	E_SequenceState.State_Active:
		//ProcessingQueue einmal durchlaufen
		fbProcessingQueue.M_SetCurrentToHead();
		REPEAT
			pStep := fbProcessingQueue.M_Get();
			IF pStep > 0 THEN
				CASE pStep^.eState OF
					E_StepState.STEPSTATUS_InQueue:
						nInfo := 0;
						//sind alle Bedingungen für eine Ausführung erfüllt?
						pStep^.bActionResultIsValid := FALSE;
						IF pStep^.pCondi > 0 THEN
							nCondiCheckResult := pStep^.pCondi^.M_Check(1);
							IF nCondiCheckResult.0 THEN
								//Hier checken, ob die Action einen Move mit Pipette beinhaltet
								//Wenn ja, dann checken, ob ZSensor mounted -> entsprechend Interaktion senden
								IF nCondiCheckResult.1 THEN //Cancel (Vergleich CondiStepResult negativ)
									//Step aus ProcessingQueue entfernen
									pStep^.bFollowerInQueue := FALSE;
									fbProcessingQueue.M_Remove(pStep);
									M_ChangeStepState(pStep, E_StepState.STEPSTATUS_Idle);
									fbSequenceInfo.M_AddTail(nId,eCurrentState,pStep);
								ELSE
									IF pStep^.stActionData.eAction = E_Action.ACTION_CounterStep THEN
										IF NOT pStep^.bFollowerInQueue THEN	//Follower in ProcessingQueue eintragen
											pStep^.bFollowerInQueue := TRUE;
											REPEAT
												pFollowStep := M_ReadFollowerStep(pStep);
												IF pFollowStep > 0 THEN
													fbProcessingQueue.M_Add(pFollowStep);
													M_ChangeStepState(pFollowStep,E_StepState.STEPSTATUS_InQueue);
													M_ChangeStepInfo(pFollowStep,0);
													fbSequenceInfo.M_AddTail(nId,eCurrentState,pFollowStep);
												END_IF
											UNTIL (pFollowStep = 0)
											END_REPEAT
										END_IF
										
										IF pStep^.stActionData.aParams[1] = 0 THEN //Set
											pStep^.nActionResult := pStep^.stActionData.aParams[2];
										ELSIF pStep^.stActionData.aParams[1] = 1 THEN //Add
											pStep^.nActionResult := pStep^.nActionResult + pStep^.stActionData.aParams[2];
										END_IF
										
										//Provisorium
										nCounter := pStep^.nActionResult;
										//Provisorium
										
										nInfo := pStep^.nActionResult;
										pStep^.bActionResultIsValid := TRUE;
										//Step aus ProcessingQueue entfernen
										pStep^.bFollowerInQueue := FALSE;
										fbProcessingQueue.M_Remove(pStep);
										M_ChangeStepState(pStep, E_StepState.STEPSTATUS_Ready);
										M_ChangeStepInfo(pStep,pStep^.nActionResult);
										fbSequenceInfo.M_AddTail(nId,eCurrentState,pStep);
									ELSIF pStep^.stActionData.eAction = E_Action.ACTION_PauseStep THEN //PauseStep führt keine Action aus
										M_ChangeStepState(pStep, E_StepState.STEPSTATUS_Active);
										fbSequenceInfo.M_AddTail(nId,eCurrentState,pStep);
									ELSE //Action ausführen
										M_ChangeStepState(pStep, E_StepState.STEPSTATUS_Active);
										IF pStep^.stActionData.eAction = E_Action.ACTION_MoveToTarget AND pStep^.stActionData.aParams[1] = E_TargetRef.TARGETREF_SequParaToArrayItem THEN
											pStep^.stActionData.aParams[2] := nSequParam;
										ELSIF pStep^.stActionData.eAction = E_Action.ACTION_RunSequence THEN
											pStep^.stActionData.aParams[2] := nCounter;
										END_IF
										stError.ErrorId := ActionDispacher.M_ExeAction(pStep^.stActionData, FALSE, nActionId=>pStep^.nActionId);
										fbSequenceInfo.M_AddTail(nId,eCurrentState,pStep);
									END_IF
								END_IF
							END_IF
						ELSE	//Step hat keine Condi
							M_ChangeStepState(pStep, E_StepState.STEPSTATUS_Active);
							IF pStep^.stActionData.eAction = E_Action.ACTION_CounterStep THEN
								IF NOT pStep^.bFollowerInQueue THEN	//Follower in ProcessingQueue eintragen
									pStep^.bFollowerInQueue := TRUE;
									REPEAT
										pFollowStep := M_ReadFollowerStep(pStep);
										IF pFollowStep > 0 THEN
											fbProcessingQueue.M_Add(pFollowStep);
											M_ChangeStepState(pFollowStep, E_StepState.STEPSTATUS_InQueue);
											M_ChangeStepInfo(pFollowStep,0);
											fbSequenceInfo.M_AddTail(nId,eCurrentState,pFollowStep);
										END_IF
									UNTIL (pFollowStep = 0)
									END_REPEAT
								END_IF
								
								IF pStep^.stActionData.aParams[1] = 0 THEN //Set
									pStep^.nActionResult := pStep^.stActionData.aParams[2];
								ELSIF pStep^.stActionData.aParams[1] = 1 THEN //Add
									pStep^.nActionResult := pStep^.nActionResult + pStep^.stActionData.aParams[2];
								END_IF
								
								//Provisorium
								nCounter := pStep^.nActionResult;
								//Provisorium
								
								pStep^.bActionResultIsValid := TRUE;
								//Step aus ProcessingQueue entfernen
								pStep^.bFollowerInQueue := FALSE;
								fbProcessingQueue.M_Remove(pStep);
								M_ChangeStepState(pStep, E_StepState.STEPSTATUS_Ready);
								M_ChangeStepInfo(pStep,pStep^.nActionResult);
								fbSequenceInfo.M_AddTail(nId,eCurrentState,pStep);
							ELSIF pStep^.stActionData.eAction = E_Action.ACTION_PauseStep THEN //PauseStep führt keine Action aus
								M_ChangeStepState(pStep, E_StepState.STEPSTATUS_Active);
								fbSequenceInfo.M_AddTail(nId,eCurrentState,pStep);
							ELSE //Action ausführen
								M_ChangeStepState(pStep, E_StepState.STEPSTATUS_Active);
								
								IF pStep^.stActionData.eAction = E_Action.ACTION_MoveToTarget AND pStep^.stActionData.aParams[1] = E_TargetRef.TARGETREF_SequParaToArrayItem THEN
									pStep^.stActionData.aParams[2] := nSequParam;
								ELSIF pStep^.stActionData.eAction = E_Action.ACTION_RunSequence THEN
									pStep^.stActionData.aParams[2] := nCounter;
								END_IF
								
								stError.ErrorId := ActionDispacher.M_ExeAction(pStep^.stActionData, FALSE, nActionId=>pStep^.nActionId);
								fbSequenceInfo.M_AddTail(nId,eCurrentState,pStep);
							END_IF
						END_IF
						
						IF stError.ErrorId > 0 THEN
							M_ChangeStepState(pStep, E_StepState.STEPSTATUS_Error);
							fbSequenceInfo.M_AddTail(nId,eCurrentState,pStep);
							bError := TRUE;
						END_IF
						
						
					E_StepState.STEPSTATUS_Active:
						IF NOT pStep^.bFollowerInQueue THEN	//Follower in ProcessingQueue eintragen
							pStep^.bFollowerInQueue := TRUE;
							REPEAT
								pFollowStep := M_ReadFollowerStep(pStep);
								IF pFollowStep > 0 THEN
									fbProcessingQueue.M_Add(pFollowStep);
									M_ChangeStepState(pFollowStep, E_StepState.STEPSTATUS_InQueue);
									M_ChangeStepInfo(pFollowStep,pFollowStep^.nActionResult);
									fbSequenceInfo.M_AddTail(nId,eCurrentState,pFollowStep);
								END_IF
							UNTIL (pFollowStep = 0)
							END_REPEAT
						END_IF
						
						IF pStep^.stActionData.eAction = E_Action.ACTION_PauseStep THEN
							eCurrentState := E_SequenceState.State_PauseRequest;
							EXIT;
						ELSE
							//Action-Status abfragen
							IF nId = 1 THEN
								nId := 1;
							END_IF
							eActionStatus := ActionDispacher.M_GetActionStatus(pStep^.nActionId,nProgress=>nInfo);
							M_ChangeStepInfo(pStep, nInfo); 
							IF eActionStatus = E_ActionStatus.ACTIONSTATUS_Ready OR eActionStatus = E_ActionStatus.ACTIONSTATUS_Idle THEN //Action nicht mehr aktiv
								//Es gibt momentan genau eine Action, welche nach ihrer Abarbeitung die Sequence in Pause versetzt (DispenseTest)
								//Rückmeldung aus ActionDispacher
								//PauseRequest beim ActionDispacher gesetzt?
								//Delay bis Fertigmeldung
								M_ChangeStepState(pStep, E_StepState.STEPSTATUS_Ready);
								pStep^.bFollowerInQueue := FALSE;
								fbProcessingQueue.M_Remove(pStep);
								IF ActionDispacher.P_bLastActionResult THEN
									pStep^.bActionResultIsValid := TRUE;
									pStep^.nActionResult := ActionDispacher.P_nLastActionResult;
									M_ChangeStepInfo(pStep, pStep^.nActionResult);
									ActionDispacher.P_bLastActionResult := FALSE;
								END_IF
								IF ActionDispacher.P_bPauseRequestIntern THEN
									ActionDispacher.P_bPauseRequestIntern := FALSE;
									eCurrentState := E_SequenceState.State_PauseRequest;
									fbSequenceInfo.M_AddTail(nId,eCurrentState,pStep);
									EXIT;
								END_IF
							ELSIF eActionStatus = E_ActionStatus.ACTIONSTATUS_Pause THEN
								//Tritt auf, wenn Action intern auf Pause gesetzt werden (z.B. Untersequenzen, welche einen Pause-Step beinhalten)
								//->Seq. selber in Pause versetzen
								M_ChangeStepState(pStep, E_StepState.STEPSTATUS_Pause);
								eCurrentState := E_SequenceState.State_Pause;
								fbSequenceInfo.M_AddTail(nId,eCurrentState,pStep);
								EXIT;
							ELSIF eActionStatus = E_ActionStatus.ACTIONSTATUS_Error THEN //Action hat Error verursacht
								M_ChangeStepState(pStep, E_StepState.STEPSTATUS_Error);
								fbProcessingQueue.M_Remove(pStep);
								bError := TRUE;
							END_IF
							//Nur melden, wenn sich am jeweiligem Step etwas geändert hat
							//Diese Info kann nur im Step selber stehen.
							fbSequenceInfo.M_AddTail(nId,eCurrentState,pStep);
						END_IF
				END_CASE
			END_IF
		UNTIL (pStep = 0)
		END_REPEAT
		//Sequence ist abgearbeitet, wenn der letzte Step ready
		IF fbProcessingQueue.P_bEmpty THEN
			eCurrentState := E_SequenceState.State_Ready;
		END_IF
		
	E_SequenceState.State_PauseRequest:
		eCurrentState := E_SequenceState.State_Pause;
		//Active Steps in PauseRequest setzen
		//In diesem State wird solange verharrt, bis kein Step mehr in Active
		//ProcessingQueue einmal durchlaufen
		fbProcessingQueue.M_SetCurrentToHead();
		REPEAT
			pStep := fbProcessingQueue.M_Get();
			IF pStep > 0 THEN
				IF pStep^.eState = E_StepState.STEPSTATUS_Active THEN
					eCurrentState := E_SequenceState.State_PauseRequest; 
					CASE ActionDispacher.M_GetActionStatus(pStep^.nActionId,nProgress=>nInfo) OF
						E_ActionStatus.ACTIONSTATUS_Active:
							ActionDispacher.M_PauseAction(pStep^.nActionId);
						E_ActionStatus.ACTIONSTATUS_Pause:
							M_ChangeStepState(pStep, E_StepState.STEPSTATUS_Pause);
							fbSequenceInfo.M_AddTail(nId,eCurrentState,pStep);
						E_ActionStatus.ACTIONSTATUS_Ready:
							M_ChangeStepState(pStep, E_StepState.STEPSTATUS_Ready);
							pStep^.bFollowerInQueue := FALSE;
							fbProcessingQueue.M_Remove(pStep);
							fbSequenceInfo.M_AddTail(nId,eCurrentState,pStep);
							IF ActionDispacher.P_bLastActionResult THEN
								pStep^.bActionResultIsValid := TRUE;
								pStep^.nActionResult := ActionDispacher.P_nLastActionResult; 
								ActionDispacher.P_bLastActionResult := FALSE;
							END_IF
					END_CASE
				END_IF
			END_IF
		UNTIL (pStep = 0)
		END_REPEAT
	E_SequenceState.State_Pause:
		//Do nothing
	E_SequenceState.State_Continue:
		//Steps, die in Pause sind, fortsetzen
		fbProcessingQueue.M_SetCurrentToHead();
		REPEAT
			pStep := fbProcessingQueue.M_Get();
			IF pStep > 0 THEN
				IF pStep^.eState = E_StepState.STEPSTATUS_Pause THEN
					ActionDispacher.M_ContinueAction(pStep^.nActionId,nProgress=>nInfo);
					M_ChangeStepState(pStep, E_StepState.STEPSTATUS_Active);
					M_ChangeStepInfo(pStep, nInfo);
					fbSequenceInfo.M_AddTail(nId,eCurrentState,pStep);
				END_IF
			END_IF
		UNTIL (pStep = 0)
		END_REPEAT
		eCurrentState := E_SequenceState.State_Active;
	
	E_SequenceState.State_Ready:
		//Do nothing
	E_SequenceState.State_Cancel:
		//Alle aktiven Steps abbrechen
		//ProcessingQueue leeren
		//in Canceled gehen
		IF nCancelState = 0 THEN
			fbComplexAction.P_nDispenseTrials := 0;
			fbProcessingQueue.M_SetCurrentToHead();
			REPEAT
				pStep := fbProcessingQueue.M_Get();
				IF pStep > 0 THEN
					IF pStep^.eState = E_StepState.STEPSTATUS_Active OR pStep^.eState = E_StepState.STEPSTATUS_Pause THEN
						ActionDispacher.M_StopAction(pStep^.nActionId);
					END_IF
				END_IF
			UNTIL (pStep = 0)
			END_REPEAT
			nCancelState := 1;
		ELSIF nCancelState = 1 THEN
			eCurrentState := E_SequenceState.State_Canceled;	
			fbProcessingQueue.M_SetCurrentToHead();
			REPEAT
				pStep := fbProcessingQueue.M_Get();
				IF pStep > 0 THEN
					IF pStep^.eState = E_StepState.STEPSTATUS_Active OR pStep^.eState = E_StepState.STEPSTATUS_Pause THEN
						//kommt man hier an?
						//geht ActionStatus in Ready oder Idle?
						//eventuell mit Scope aufzeichnen
						IF ActionDispacher.M_GetActionStatus(pStep^.nActionId) <> E_ActionStatus.ACTIONSTATUS_Ready THEN
							eCurrentState := E_SequenceState.State_Cancel;
						END_IF
					END_IF
				END_IF
			UNTIL (pStep = 0)
			END_REPEAT			
		END_IF
END_CASE

IF eOldState <> eCurrentState THEN
	//Progress?
	fbSequenceInfo.M_AddTail(nId,eCurrentState,0);
	eOldState := eCurrentState;
END_IF

IF bError THEN
	fbComplexAction.P_nDispenseTrials := 0;
	stError.POU := POU_FB_Sequenece;
	fbErrorList.M_Add(stError);
	eCurrentState := E_SequenceState.State_Error;
	bError := FALSE;
END_IF

METHOD FB_init : BOOL
VAR_INPUT
	bInitRetains : BOOL; // if TRUE, the retain variables are initialized (warm start / cold start)
	bInCopyCode : BOOL;  // if TRUE, the instance afterwards gets moved into the copy code (online change)
	nNoOfSteps	: UINT;
END_VAR
fbStepList.FB_SetNoOfSteps(nNoOfSteps);
END_METHOD

METHOD M_AddCondi : ERRORID
VAR_INPUT
	refCmdData : REFERENCE TO  ST_CmdData;	
END_VAR
VAR
	eOperator : E_LogicOperator;
	pCondi : POINTER TO FB_CondiBase;
	pStep  : POINTER TO ST_Step; 
END_VAR
//checken, ob zugehörige /ProgramNr/StepNr vorhanden, dh. es muss schon eine Condition vorhanden sein, in die dann der
//Zeiger auf hinzuzufügende Condition eingetragen wird
pStep := fbStepList.M_Get(refCmdData.aHeader[0]);
IF pStep = 0 THEN
	M_AddCondi := E_ErrorIdCmd.ERRORID_StepNotExists;
	RETURN;
END_IF

IF pStep^.pCondi = 0 THEN	//Step besitzt noch keine Condition und kann deshalb keine zusätzliche bekommen
	M_AddCondi := E_ErrorIdCmd.ERRORID_StepHasNoBasicCondi;
	RETURN;
END_IF

eOperator := UINT_TO_USINT(refCmdData.aHeader[1]);

IF NOT (eOperator = E_LogicOperator.LOGIC_OP_AND OR eOperator = E_LogicOperator.LOGIC_OP_OR) THEN	//unzulässiger CondiOperator
	M_AddCondi := E_ErrorIdCmd.ERRORID_InvalidCondiOperator;
	RETURN;
END_IF

M_AddCondi := M_CreateCondi(pStep:= pStep, 
				eOperator:= eOperator, 
				eCondition:= DINT_TO_USINT(refCmdData.n32Data[0]), 
				nValue1:= refCmdData.n32Data[1], 
				nValue2:= refCmdData.n32Data[2], 
				nValue3:= refCmdData.n32Data[3], 
				pCondi=>pCondi);

IF M_AddCondi = 0 THEN
	pStep^.pCondi^.M_AddNext(pCondi);
END_IF
END_METHOD

METHOD M_AddStep : ERRORID
VAR_INPUT
	refCmdData : REFERENCE TO  ST_CmdData;
END_VAR

VAR
	stStep		: ST_Step;
	eCondition 	: E_Condition;
END_VAR
//Es werden nur Programmsätze mit zulässiger Action hinzugefügt
stStep.nStepNr := refCmdData.aHeader[0];
stStep.bStop := refCmdData.aHeader[1].0;
stStep.tDelay := UINT_TO_TIME(refCmdData.aHeader[2]);
stStep.stActionData.eAction := DINT_TO_UINT(refCmdData.n32Data[5]);
stStep.stActionData.nObject := DINT_TO_UINT(refCmdData.n32Data[6]);
stStep.bFollowerInQueue := FALSE;
stStep.bHasForerunner := FALSE;

//Basiscondtion hinzufügen
eCondition := DINT_TO_USINT(refCmdData.n32Data[0]);

M_AddStep := M_CreateCondi(pStep:= ADR(stStep), 
							eOperator:= E_LogicOperator.LOGIC_OP_AND,	//bei der ersten Condi immer "AND"
							eCondition:= eCondition, 
							nValue1:= refCmdData.n32Data[1], 
							nValue2:= refCmdData.n32Data[2], 
							nValue3:= refCmdData.n32Data[3], 
							pCondi=> stStep.pCondi);

IF M_AddStep > 0 THEN
	RETURN;
END_IF

CASE stStep.stActionData.eAction OF
	//BasicActions
	E_Action.ACTION_MoveXY, E_Action.ACTION_MoveZ, E_Action.ACTION_SetPressure, E_Action.ACTION_SetVacuum, E_Action.ACTION_SwitchPressure, 
	E_Action.ACTION_Heating, E_Action.ACTION_Cooling, E_Action.ACTION_Aspirate, E_Action.ACTION_Dispense, E_Action.ACTION_DispenseDrops, 
	E_Action.ACTION_InkSpin, E_Action.ACTION_Expose, E_Action.ACTION_InkOpClCover, E_Action.ACTION_ReactorOpCl, E_Action.ACTION_FillLiquid,
	E_Action.ACTION_EmptyLiquid, E_Action.ACTION_DilPrepare,E_Action.ACTION_Mix,E_Action.ACTION_MeasurepH,E_Action.ACTION_SetVoltage,
	E_Action.ACTION_SuckOff, E_Action.ACTION_BasicDispense, E_Action.ACTION_StirrCartridge,
	E_Action.ACTION_MoveLifter, E_Action.ACTION_TurnTo:
		//max 8 Parameter kopieren
		MEMCPY(ADR(stStep.stActionData.aParams),ADR(refCmdData.n32Data[7]),32);
	E_Action.ACTION_TakePicture:
		//1 Parameter kopieren
		MEMCPY(ADR(stStep.stActionData.aParams),ADR(refCmdData.n32Data[7]),4);
		//Parameter 2 wird mit SequenceID gefüllt und Parameter 3 wird mit StepNummer gefüllt
		stStep.stActionData.aParams[2] := UDINT_TO_DINT(nId);
		stStep.stActionData.aParams[3] := stStep.nStepNr;
	
	//ComplexActions
	E_Action.ACTION_MoveToTarget, E_Action.ACTION_ExchangePiece,E_Action.ACTION_OpenCloseFlipTube,E_Action.ACTION_InsertTool,
	E_Action.ACTION_DockTool:
		//Object muss ein MzTool sein
		IF fbObjectDirectory.M_ObjIsMzTool(stStep.stActionData.nObject) THEN
			stStep.stActionData.nTarget := DINT_TO_UINT(refCmdData.n32Data[7]);
			//Target checken
			IF fbObjectDirectory.M_ObjIsTarget(stStep.stActionData.nTarget) THEN
				//11 Parameter kopieren
				MEMCPY(ADR(stStep.stActionData.aParams),ADR(refCmdData.n32Data[8]),44);
			ELSE
				M_AddStep := E_ErrorIdCmd.ERRORID_UnsuitableTarget;
			END_IF
		ELSE
			M_AddStep := E_ErrorIdCmd.ERRORID_UnsuitableObject;
		END_IF

	E_Action.ACTION_TransferGas, E_Action.ACTION_TransferLiquid:
		//Object und Target müssen ein Luers sein
		IF fbObjectDirectory.M_GetObjType(stStep.stActionData.nObject) = E_ObjectType.OBJECTTYPE_Luer THEN
			stStep.stActionData.nTarget := DINT_TO_UINT(refCmdData.n32Data[7]);
			IF fbObjectDirectory.M_GetObjType(stStep.stActionData.nTarget) = E_ObjectType.OBJECTTYPE_Luer THEN
				//max. 3 Parameter kopieren
				MEMCPY(ADR(stStep.stActionData.aParams),ADR(refCmdData.n32Data[8]),12);
			ELSE
				M_AddStep := E_ErrorIdCmd.ERRORID_UnsuitableObject;
			END_IF
		ELSE
			M_AddStep := E_ErrorIdCmd.ERRORID_UnsuitableObject;
		END_IF
		
	E_Action.ACTION_TransferTray:
		IF fbObjectDirectory.M_ObjIsDevice(stStep.stActionData.nObject) THEN
			MEMCPY(ADR(stStep.stActionData.aParams),ADR(refCmdData.n32Data[8]),4);
		ELSE
			M_AddStep := E_ErrorIdCmd.ERRORID_UnsuitableObject;
		END_IF
	
	E_Action.ACTION_MeasureTool:
		//Object muss ein MzTool sein
		IF fbObjectDirectory.M_ObjIsMzTool(stStep.stActionData.nObject) THEN
			stStep.stActionData.nTarget := DINT_TO_UINT(refCmdData.n32Data[7]);
			MEMCPY(ADR(stStep.stActionData.aParams),ADR(refCmdData.n32Data[8]),12);
			//Target checken
			IF fbObjectDirectory.M_ObjIsTarget(stStep.stActionData.nTarget) THEN
				;
			ELSE
				M_AddStep := E_ErrorIdCmd.ERRORID_UnsuitableTarget;
			END_IF
		ELSE
			M_AddStep := E_ErrorIdCmd.ERRORID_UnsuitableObject;
		END_IF		
		
	E_Action.ACTION_CleanTip:
		//Object muss ein MzTool sein
		IF fbObjectDirectory.M_ObjIsMzTool(stStep.stActionData.nObject) THEN
			stStep.stActionData.nTarget := DINT_TO_UINT(refCmdData.n32Data[7]);
			//Target checken
			IF fbObjectDirectory.M_GetObjType(stStep.stActionData.nTarget) = E_ObjectType.OBJECTTYPE_TipCleaner THEN
				;
			ELSIF
				fbObjectDirectory.M_GetObjType(stStep.stActionData.nTarget) = E_ObjectType.OBJECTTYPE_TipCleanerGen2 THEN
				MEMCPY(ADR(stStep.stActionData.aParams[1]),ADR(refCmdData.n32Data[8]),16);
			ELSE
				M_AddStep := E_ErrorIdCmd.ERRORID_UnsuitableTarget;
			END_IF
		ELSE
			M_AddStep := E_ErrorIdCmd.ERRORID_UnsuitableObject;
		END_IF
		
	E_Action.ACTION_DryPip:
		//Object muss ein MzTool sein
		IF fbObjectDirectory.M_ObjIsMzTool(stStep.stActionData.nObject) THEN
			stStep.stActionData.nTarget := DINT_TO_UINT(refCmdData.n32Data[7]);
			//Target checken
			IF fbObjectDirectory.M_GetObjType(stStep.stActionData.nTarget) = E_ObjectType.OBJECTTYPE_DryPad THEN
				MEMCPY(ADR(stStep.stActionData.aParams[1]),ADR(refCmdData.n32Data[8]),8);
			ELSE
				M_AddStep := E_ErrorIdCmd.ERRORID_UnsuitableTarget;
			END_IF
		ELSE
			M_AddStep := E_ErrorIdCmd.ERRORID_UnsuitableObject;
		END_IF		
		
	E_Action.ACTION_WashTool:
		//Object muss eine Pipette sein
		IF fbObjectDirectory.M_GetObjType(stStep.stActionData.nObject) = E_ObjectType.OBJECTTYPE_PiezoPip OR
				fbObjectDirectory.M_GetObjType(stStep.stActionData.nObject) = E_ObjectType.OBJECTTYPE_PassivPip OR
				fbObjectDirectory.M_GetObjType(stStep.stActionData.nObject) = E_ObjectType.OBJECTTYPE_Luer OR
				fbObjectDirectory.M_GetObjType(stStep.stActionData.nObject) = E_ObjectType.OBJECTTYPE_SolenoidPip OR
				fbObjectDirectory.M_GetObjType(stStep.stActionData.nObject) = E_ObjectType.OBJECTTYPE_TitrationTool OR
				fbObjectDirectory.M_GetObjType(stStep.stActionData.nObject) = E_ObjectType.OBJECTTYPE_TwinPiezoHolder OR
				fbObjectDirectory.M_GetObjType(stStep.stActionData.nObject) = E_ObjectType.OBJECTTYPE_TriplePip THEN
			stStep.stActionData.nTarget := DINT_TO_UINT(refCmdData.n32Data[7]);
			//Target checken
			IF fbObjectDirectory.M_GetObjType(stStep.stActionData.nTarget) = E_ObjectType.OBJECTTYPE_WashStation THEN
				//5 Parameter kopieren
				MEMCPY(ADR(stStep.stActionData.aParams[1]),ADR(refCmdData.n32Data[8]),60);
			ELSE
				M_AddStep := E_ErrorIdCmd.ERRORID_UnsuitableTarget;
			END_IF
		ELSE
			M_AddStep := E_ErrorIdCmd.ERRORID_UnsuitableObject;
		END_IF
		
	E_Action.ACTION_DispenseTest:
		//Object muss eine PiezoPip
		IF (fbObjectDirectory.M_GetObjType(stStep.stActionData.nObject) = E_ObjectType.OBJECTTYPE_PiezoPip) OR
			(fbObjectDirectory.M_GetObjType(stStep.stActionData.nObject) = E_ObjectType.OBJECTTYPE_TwinPiezoHolder) THEN
			stStep.stActionData.nTarget := DINT_TO_UINT(refCmdData.n32Data[7]);
			//Target checken
			IF fbObjectDirectory.M_GetObjType(stStep.stActionData.nTarget) = E_ObjectType.OBJECTTYPE_Stroboscope THEN
				MEMCPY(ADR(stStep.stActionData.aParams[1]),ADR(refCmdData.n32Data[8]),8);
			ELSE
				M_AddStep := E_ErrorIdCmd.ERRORID_UnsuitableTarget;
			END_IF
		ELSE
			M_AddStep := E_ErrorIdCmd.ERRORID_UnsuitableObject;
		END_IF

	E_Action.ACTION_GetPipSample:
		//Object muss eine Pipette sein
		IF fbObjectDirectory.M_GetObjType(stStep.stActionData.nObject) = E_ObjectType.OBJECTTYPE_PiezoPip OR
				fbObjectDirectory.M_GetObjType(stStep.stActionData.nObject) = E_ObjectType.OBJECTTYPE_PassivPip OR
				fbObjectDirectory.M_GetObjType(stStep.stActionData.nObject) = E_ObjectType.OBJECTTYPE_SolenoidPip OR
				fbObjectDirectory.M_GetObjType(stStep.stActionData.nObject) = E_ObjectType.OBJECTTYPE_TwinPiezoHolder THEN
			stStep.stActionData.nTarget := DINT_TO_UINT(refCmdData.n32Data[7]);
			//Target checken
			IF fbObjectDirectory.M_GetObjType(stStep.stActionData.nTarget) = E_ObjectType.OBJECTTYPE_Mtp THEN
				//6 Parameter kopieren
				MEMCPY(ADR(stStep.stActionData.aParams[1]),ADR(refCmdData.n32Data[8]),24);		
			ELSE
				M_AddStep := E_ErrorIdCmd.ERRORID_UnsuitableTarget;
			END_IF
		ELSE
			M_AddStep := E_ErrorIdCmd.ERRORID_UnsuitableObject;
		END_IF
		
	E_Action.ACTION_StampDemolding:
		//Object muss ein StampSupport sein
		IF fbObjectDirectory.M_GetObjType(stStep.stActionData.nObject) = E_ObjectType.OBJECTTYPE_StampSupport THEN
			//6 Parameter kopieren
			MEMCPY(ADR(stStep.stActionData.aParams[1]),ADR(refCmdData.n32Data[7]),24);			
		ELSE
			M_AddStep := E_ErrorIdCmd.ERRORID_UnsuitableObject;
		END_IF
		
	E_Action.ACTION_StampInking:
		//Object muss ein StampSupport sein
		IF fbObjectDirectory.M_GetObjType(stStep.stActionData.nObject) = E_ObjectType.OBJECTTYPE_StampSupport THEN
			stStep.stActionData.nTarget := DINT_TO_UINT(refCmdData.n32Data[7]);
			//3 Parameter kopieren
			MEMCPY(ADR(stStep.stActionData.aParams[1]),ADR(refCmdData.n32Data[8]),12);
		ELSE	
			M_AddStep := E_ErrorIdCmd.ERRORID_UnsuitableObject;
		END_IF
		
	E_Action.ACTION_PickPutPowder:
		//Object kann nur eine Pulverpipette sein
		IF fbObjectDirectory.M_GetObjType(stStep.stActionData.nObject) = E_ObjectType.OBJECTTYPE_PowderPip OR
			fbObjectDirectory.M_GetObjType(stStep.stActionData.nObject) = E_ObjectType.OBJECTTYPE_PickPlacePip THEN
			//7 Parameter kopieren
			MEMCPY(ADR(stStep.stActionData.aParams[1]),ADR(refCmdData.n32Data[7]),28);		
		ELSE
			M_AddStep := E_ErrorIdCmd.ERRORID_UnsuitableObject;
		END_IF

	E_Action.ACTION_PowdStatShaking:
		//Object kann nur eine PowderStation sein
		IF fbObjectDirectory.M_GetObjType(stStep.stActionData.nObject) = E_ObjectType.OBJECTTYPE_PowderStation THEN
			//5 Parameter kopieren
			MEMCPY(ADR(stStep.stActionData.aParams[1]),ADR(refCmdData.n32Data[7]),20);		
		ELSE
			M_AddStep := E_ErrorIdCmd.ERRORID_UnsuitableObject;
		END_IF
	
	E_Action.ACTION_PowdStatLeveling:		
		//Object kann nur eine PowderStation sein
		IF fbObjectDirectory.M_GetObjType(stStep.stActionData.nObject) = E_ObjectType.OBJECTTYPE_PowderStation THEN
			stStep.stActionData.aParams[1] := (refCmdData.n32Data[7]);
		ELSE
			M_AddStep := E_ErrorIdCmd.ERRORID_UnsuitableObject;
		END_IF
		
	E_Action.ACTION_ActionOnArray:
		//Object muss ein MzTool sein
		IF fbObjectDirectory.M_ObjIsMzTool(stStep.stActionData.nObject) THEN
			stStep.stActionData.nTarget := DINT_TO_UINT(refCmdData.n32Data[7]);
			//Target checken
			IF fbObjectDirectory.M_ObjIsArray(stStep.stActionData.nTarget) THEN 
				//18 Parameter kopieren
				MEMCPY(ADR(stStep.stActionData.aParams),ADR(refCmdData.n32Data[8]),72);
				//Wenn Action TakePicture, dann SequenceID und StepNummer übertragen
				IF stStep.stActionData.aParams[11] = E_Action.ACTION_TakePicture THEN
					//stStep.stActionData.aParams[12] = Delay
					stStep.stActionData.aParams[13] := UDINT_TO_DINT(nId);
					stStep.stActionData.aParams[14] := stStep.nStepNr;
				END_IF
			ELSE
				M_AddStep := E_ErrorIdCmd.ERRORID_UnsuitableTarget;
			END_IF
		ELSE
			M_AddStep := E_ErrorIdCmd.ERRORID_UnsuitableObject;
		END_IF
		
	E_Action.ACTION_RunGCode:
			//6 Parameter kopieren
			stStep.stActionData.nTarget := DINT_TO_UINT(refCmdData.n32Data[6]);
			MEMCPY(ADR(stStep.stActionData.aParams[1]),ADR(refCmdData.n32Data[7]),52);
	E_Action.ACTION_Delay, E_Action.ACTION_CoupleHeads:
			stStep.stActionData.aParams[1] := refCmdData.n32Data[6];
	E_Action.ACTION_RunSequence:
			MEMCPY(ADR(stStep.stActionData.aParams[1]),ADR(refCmdData.n32Data[6]),24);
			IF DINT_TO_UDINT(stStep.stActionData.aParams[1]) = nId THEN
				M_AddStep := E_ErrorIdCmd.ERRORID_SequenceCannotCallItself;
			ELSE
				//Sequence vorhanden?
				IF fbSequenceList.M_Get(DINT_TO_UDINT(stStep.stActionData.aParams[1])) = 0 THEN
					M_AddStep := E_ErrorIdCmd.ERRORID_SequenceNotExists;
				END_IF
			END_IF
	E_Action.ACTION_GoToStep:
			//Follower eintragen
			M_AddStep := F_SetFollowerStep(ADR(stStep),DINT_TO_UINT(refCmdData.n32Data[6]));
	E_Action.ACTION_CounterStep:
			stStep.stActionData.aParams[1] := refCmdData.n32Data[6]; //Operator (0=set, 1=Add)
			stStep.stActionData.aParams[2] := refCmdData.n32Data[7]; //Amount
			
	E_Action.ACTION_PauseStep:
		;
	ELSE
		M_AddStep := E_ErrorIdCmd.ERRORID_InvalidAction;
END_CASE

IF M_AddStep > 0 THEN	//Condition wieder löschen!!
	__DELETE(stStep.pCondi);
ELSE
	M_AddStep := fbStepList.M_Add(stStep);
	IF M_AddStep > 0 THEN
		__DELETE(stStep.pCondi);
	END_IF
END_IF
END_METHOD

METHOD M_ChangeStepInfo
VAR_INPUT
	pStep : POINTER TO ST_Step;
	nInfo : DINT;
END_VAR
IF pStep^.nInfo <> nInfo THEN
	pStep^.nInfo := nInfo;
	pStep^.bInfoChanged := TRUE;
END_IF
END_METHOD

METHOD M_ChangeStepState
VAR_INPUT
	pStep : POINTER TO ST_Step;
	eState : E_StepState;
END_VAR
IF pStep^.eState = eState THEN
	RETURN;
END_IF
//Übergänge
// von "active" nach "ready" -> stepsReady inkrementieren
// von "ready" nach "InQueue"  -> stepsReady dekrementieren
// von allen States nach "Idle" -> stepsReady dekrementieren
IF pStep^.eState = E_StepState.STEPSTATUS_Active AND eState = E_StepState.STEPSTATUS_Ready THEN
	nStepsReady := MIN(fbStepList.P_nCount,nStepsReady + 1);
ELSIF (pStep^.eState = E_StepState.STEPSTATUS_Ready AND eState = E_StepState.STEPSTATUS_InQueue) OR
 		eState = E_StepState.STEPSTATUS_Idle THEN
	IF nStepsReady > 0 THEN	//Vermeiden, dass negativee Überlauf bei Neustart der Sequenz stattfindet
		nStepsReady := nStepsReady - 1;	
	END_IF
END_IF
pStep^.eState := eState;
pStep^.bInfoChanged := TRUE;
END_METHOD

METHOD M_CheckForStart : ERRORID
VAR_INPUT
END_VAR
IF fbStepList.P_nCount = 0 THEN
	M_CheckForStart := E_ErrorIdCmd.ERRORID_NoStepsInSequence;
	RETURN;
END_IF

IF NOT eCurrentState = E_SequenceState.State_Idle THEN
	M_CheckForStart := E_ErrorIdCmd.ERRORID_InvalidState;
	RETURN;
END_IF
END_METHOD

METHOD M_Continue : ERRORID
VAR_INPUT
END_VAR
IF eCurrentState = E_SequenceState.State_Pause THEN
	eCurrentState := E_SequenceState.State_Continue;
END_IF
END_METHOD

METHOD M_CreateCondi : ERRORID
VAR_INPUT
	pStep		: POINTER TO ST_Step;
	eOperator	: E_LogicOperator;
	eCondition 	: E_Condition;
	nValue1		: DINT;
	nValue2		: DINT;
	nValue3		: DINT;
END_VAR
VAR_OUTPUT
	pCondi	: POINTER TO FB_CondiBase;
END_VAR
VAR
	pCondiStepReady		: POINTER TO FB_CondiStepReady;
	pCondiProcessData	: POINTER TO FB_CondiProcessData;
	pCondiStepResult 	: POINTER TO FB_CondiStepResult;
	nSpecStepNr 		: UINT;
	pRefStep			: POINTER TO ST_Step;
	nDeviceObjId		: UINT;
	iDevice				: I_Device;
	eProcDataType		: E_ProcDataType;
END_VAR
IF pStep = 0 THEN
	M_CreateCondi := E_ErrorIdCmd.ERRORID_StepNotExists;
END_IF
CASE eCondition OF
	E_Condition.CONDITION_Nothing:
	;
	E_Condition.CONDITION_PreStepReady:
		//Vorgängerschritt vorhanden?
		pRefStep := fbStepList.M_Get(pStep^.nStepNr - 1);
		IF pRefStep > 0 THEN
			//Step als Follower in PreStep eintragen
			M_CreateCondi := F_SetFollowerStep(pStep:= pRefStep, pStep^.nStepNr);
			IF M_CreateCondi = 0 THEN
				pStep^.bHasForerunner := TRUE;
				pCondiStepReady := __NEW(FB_CondiStepReady);
				pCondiStepReady^.P_eOperator := eOperator;
				pCondiStepReady^.P_pStep := fbStepList.M_Get(pStep^.nStepNr - 1);
				pCondiStepReady^.P_eCondition := E_Condition.CONDITION_PreStepReady;
				pCondi := pCondiStepReady;
			END_IF
		ELSE
			M_CreateCondi := E_ErrorIdCmd.ERRORID_PrestepNotExists;
		END_IF
		
	E_Condition.CONDITION_SpecStepReady:
		//angegebener Schritt vorhanden?
		nSpecStepNr := DINT_TO_UINT(nValue1);
		pRefStep := fbStepList.M_Get(nSpecStepNr);
		IF pRefStep > 0 THEN
			//Step als Follower in PreStep eintragen
			M_CreateCondi := F_SetFollowerStep(pStep:= pRefStep,pStep^.nStepNr);
			IF M_CreateCondi = 0 THEN
				pStep^.bHasForerunner := TRUE;
				pCondiStepReady := __NEW(FB_CondiStepReady);
				pCondiStepReady^.P_eOperator := eOperator;
				pCondiStepReady^.P_pStep := fbStepList.M_Get(nSpecStepNr);
				pCondiStepReady^.P_eCondition := E_Condition.CONDITION_SpecStepReady;
				pCondi := pCondiStepReady;
			END_IF
		ELSE
			M_CreateCondi := E_ErrorIdCmd.ERRORID_SpecstepNotExists;
		END_IF
		
	E_Condition.CONDITION_ProcessVarLEQ, E_Condition.CONDITION_ProcessVarGEQ:
		//In Value2 steht das Object -> checken ob gültiges Object
		nDeviceObjId := DINT_TO_UINT(nValue2);
		IF NOT fbObjectDirectory.M_ObjIsDevice(nDeviceObjId) THEN
			M_CreateCondi := ERRORID_InvalidDeviceForProcData;
			RETURN;
		END_IF
		iDevice := fbObjectDirectory.M_GetDevice(nDeviceObjId);
		
		//In Value1 steht der Prozessdatentyp -> Checken, ob Device Daten für diesen Typ anbietet
		eProcDataType := DINT_TO_USINT(nValue1);
		IF iDevice.M_CheckProcDataType(eProcDataType) THEN
			pCondiProcessData := __NEW(FB_CondiProcessData);
			pCondiProcessData^.P_eOperator := eOperator;
			pCondiProcessData^.P_eCondition := eCondition;
			pCondiProcessData^.P_iDevice := iDevice;
			pCondiProcessData^.P_eProcDataType := eProcDataType;
			pCondiProcessData^.P_nValue := nValue3;
			pCondi := pCondiProcessData;
			
		ELSE
			M_CreateCondi := ERRORID_InvalidDeviceForProcData;
		END_IF
	E_Condition.CONDITION_StepResult:
		//angegebener Schritt vorhanden?
		nSpecStepNr := DINT_TO_UINT(nValue1);
		pRefStep := fbStepList.M_Get(nSpecStepNr);
		IF pRefStep > 0 THEN
			//Step als Follower in RefStep eintragen
			M_CreateCondi := F_SetFollowerStep(pStep:= pRefStep, pStep^.nStepNr);
			IF M_CreateCondi = 0 THEN
				pStep^.bHasForerunner := TRUE;
				pCondiStepResult := __NEW(FB_CondiStepResult);
				pCondiStepResult^.P_eCondition := eCondition;
				pCondiStepResult^.P_eOperator := eOperator;
				pCondiStepResult^.P_pStep := pRefStep;
				pCondiStepResult^.P_eCompareOperator := DINT_TO_USINT(nValue2);
				pCondiStepResult^.P_nCompareValue := nValue3;
				pCondi := pCondiStepResult;
			END_IF
		ELSE
			M_CreateCondi := E_ErrorIdCmd.ERRORID_SpecstepNotExists;
		END_IF
ELSE
	M_CreateCondi := E_ErrorIdCmd.ERRORID_InvalidCondition;
END_CASE
END_METHOD

METHOD M_Delete : BOOL
VAR_INPUT
	nMaxSteps	: UINT;
END_VAR
VAR_OUTPUT
	nDeletedSteps : UINT;
END_VAR
M_Delete := fbStepList.M_Delete(nMaxSteps:= nMaxSteps, nDeletedSteps=> nDeletedSteps);
END_METHOD

METHOD M_GetNextStep : BOOL
VAR_INPUT
END_VAR
END_METHOD

METHOD M_Pause : ERRORID
VAR_INPUT
END_VAR
IF eCurrentState = E_SequenceState.State_Active THEN
	eCurrentState := E_SequenceState.State_PauseRequest;
	//fbSequenceInfo.M_AddTail(nId,eCurrentState,0);
END_IF
END_METHOD

METHOD M_ReadFollowerStep : POINTER TO ST_Step
VAR_INPUT
	pStep : POINTER TO ST_Step;
END_VAR

VAR
	nMaxFollowers : USINT;
END_VAR

VAR_INST
	i : USINT;
END_VAR
IF pStep > 0 THEN
	nMaxFollowers := UINT_TO_USINT(SIZEOF (pStep^.aFollower) / 2);
	IF i < nMaxFollowers THEN
		IF pStep^.aFollower[i] > 0 THEN
			M_ReadFollowerStep := fbStepList.M_Get(pStep^.aFollower[i]);
			i := i + 1;
		ELSE
			i := 0;
		END_IF
	ELSE
		i := 0;
	END_IF
END_IF
END_METHOD

METHOD M_Reset
VAR_INPUT
END_VAR
IF eCurrentState = E_SequenceState.State_Error OR
	eCurrentState = E_SequenceState.State_Ready OR
	eCurrentState = E_SequenceState.State_Canceled THEN
	eCurrentState := E_SequenceState.State_Idle;
END_IF
END_METHOD

METHOD M_Start
VAR_INPUT
	nSequParam : UINT;
END_VAR
IF eCurrentState = E_SequenceState.State_Idle OR 
	eCurrentState = E_SequenceState.State_Ready OR
	eCurrentState = E_SequenceState.State_Canceled THEN
	eCurrentState := E_SequenceState.State_Start;
	nStepsReady := 0;
	THIS^.nSequParam := nSequParam;
END_IF
END_METHOD

METHOD M_Stop : BOOL
VAR_INPUT
END_VAR
IF eCurrentState = E_SequenceState.State_Active OR 
	eCurrentState = E_SequenceState.State_Pause OR eCurrentState = E_SequenceState.State_PauseRequest THEN
	eCurrentState := E_SequenceState.State_Cancel;
END_IF
END_METHOD

PROPERTY P_nCount : UINT
GET
P_nCount := fbStepList.P_nCount;
END_GET
END_PROPERTY

PROPERTY P_nId : UDINT
GET
P_nId := nId;
END_GET
SET
nId := P_nId;
END_SET
END_PROPERTY

PROPERTY P_nProgress : UINT
GET
//Gibt den Fortschritt in % an (momentan auf Anzahl abgearbeiteter Schritte bezogen)
P_nProgress := 100 * nStepsReady / fbStepList.P_nCount;
END_GET
END_PROPERTY

END_FUNCTION_BLOCK

// ---- Sequence/FB_StepList.TcPOU
{attribute 'enable_dynamic_creation'}
FUNCTION_BLOCK FB_StepList
VAR_INPUT
END_VAR
VAR_OUTPUT
END_VAR
VAR
	nStepCount	: UINT;	
	nNoOfSteps	: UINT;
	pIndexTable : POINTER TO PVOID;
END_VAR

METHOD FB_exit : BOOL
VAR_INPUT
	bInCopyCode : BOOL; // if TRUE, the exit method is called for exiting an instance that is copied afterwards (online change).
END_VAR
IF pIndexTable > 0 THEN
	__DELETE(pIndexTable);
END_IF
END_METHOD

METHOD FB_SetNoOfSteps
VAR_INPUT
	nNoOfSteps : UINT;
END_VAR

VAR
END_VAR
THIS^.nNoOfSteps := nNoOfSteps;
pIndexTable := __NEW(PVOID, nNoOfSteps);
MEMSET(pIndexTable,0,SIZEOF(PVOID) * nNoOfSteps);
END_METHOD

METHOD M_Add : ERRORID
VAR_INPUT
	stStep	: ST_STEP;
END_VAR

VAR
	pStep : POINTER TO ST_STEP;
END_VAR
//StepNr muss größer "0" sein
IF stStep.nStepNr < 1 THEN
	M_Add := E_ErrorIdCmd.ERRORID_InvalidStepNr;
	RETURN;
END_IF

//StepNr größer, als maximale Anzahl Steps beim Erstellen der Sequence angegeben
IF stStep.nStepNr > nNoOfSteps THEN
	M_Add := E_ErrorIdCmd.ERRORID_StepNrExeedsMaxNoOfSteps;
	RETURN;
END_IF

//Step existiert schon
//Das hier funzt nicht so recht.
//Es wäre hier wahrscheinlich sehr hilfreich, einen Pointer auf WORD zu definieren
IF pIndexTable[stStep.nStepNr - 1] > 0 THEN
	M_Add := E_ErrorIdCmd.ERRORID_StepAlreadyExists;
	RETURN;
END_IF

//StepNr muss immer eins größer sein als letzte Step 
IF stStep.nStepNr < nStepCount THEN
	M_Add := E_ErrorIdCmd.ERRORID_InvalidStepNr;
	RETURN;	
END_IF

pStep := __NEW(ST_STEP);
MEMCPY(pStep,ADR(stStep),SIZEOF(ST_STEP));
pIndexTable[stStep.nStepNr - 1] := pStep; 
nStepCount := nStepCount + 1;
END_METHOD

METHOD M_Delete : BOOL
VAR_INPUT
	nMaxSteps	: UINT;
END_VAR
VAR_OUTPUT
	nDeletedSteps : UINT;
END_VAR
VAR
	pStep : POINTER TO ST_STEP;
	pCondi: POINTER TO FB_CondiBase;
END_VAR

VAR_INST
	i : UINT;
END_VAR
IF pIndexTable = 0 THEN
	M_Delete := TRUE;
	RETURN;	
END_IF
//Maximal 200 Steps auf einmal löschen
WHILE i < nNoOfSteps DO
	IF pIndexTable[i] > 0 THEN
		pStep := pIndexTable[i];
		pCondi := pStep^.pCondi;
		//Condi freigeben
		IF pCondi > 0 THEN
			pCondi^.M_ClearNext();
			__DELETE(pCondi);
		END_IF
		__DELETE(pStep);
		nDeletedSteps := nDeletedSteps + 1;
		i := i + 1;
		IF nDeletedSteps = nMaxSteps THEN
			RETURN;
		END_IF		
	ELSE
		EXIT;
	END_IF
END_WHILE

i := 0;
MEMSET(pIndexTable,0,SIZEOF(DWORD) * nNoOfSteps);
nStepCount := 0;
M_Delete := TRUE;
END_METHOD

METHOD M_Get : POINTER TO ST_Step
VAR_INPUT
	nStepNr	: UINT;
END_VAR
IF nStepNr > 0 AND nStepNr <= nNoOfSteps THEN
	M_Get := pIndexTable[nStepNr - 1];
END_IF
END_METHOD

METHOD M_GetLast : POINTER TO ST_STEP
VAR_INPUT
END_VAR
IF nNoOfSteps > 0 THEN
	M_GetLast := pIndexTable[nNoOfSteps - 1];
END_IF
END_METHOD

PROPERTY P_nCount : UINT
GET
P_nCount := nStepCount;
END_GET
END_PROPERTY

END_FUNCTION_BLOCK

// ---- Sequence/FB_CondiBase.TcPOU
{attribute 'enable_dynamic_creation'}
FUNCTION_BLOCK FB_CondiBase
VAR_INPUT
END_VAR
VAR_OUTPUT
END_VAR
VAR_IN_OUT
END_VAR
VAR
	eCondition		: E_Condition;
	pNextCondi		: POINTER TO FB_CondiBase;
	eCondiOperator	: E_LogicOperator;
END_VAR

PROPERTY P_eCondition : E_Condition
SET
eCondition := P_eCondition;
END_SET
END_PROPERTY

METHOD M_ClearNext
VAR_INPUT
END_VAR
IF pNextCondi > 0 THEN
	pNextCondi^.M_ClearNext();
	__DELETE(pNextCondi);
END_IF
END_METHOD

PROPERTY P_eOperator : E_LogicOperator
SET
eCondiOperator := P_eOperator;
END_SET
END_PROPERTY

METHOD M_AddNext
VAR_INPUT
	pCondi : POINTER TO FB_CondiBase;
END_VAR
IF pNextCondi = 0 THEN
	pNextCondi := pCondi;
ELSE
	pNextCondi^.M_AddNext(pCondi);
END_IF
END_METHOD

METHOD M_Check : BYTE
VAR_INPUT
	//bPreResult	: BOOL;
	nPreResult : BYTE;
END_VAR
END_METHOD

END_FUNCTION_BLOCK

// ---- Sequence/FB_ProcessingQueue.TcPOU
FUNCTION_BLOCK FB_ProcessingQueue
VAR_INPUT
END_VAR
VAR_OUTPUT
END_VAR
VAR
	pHead	: POINTER TO ST_Pointer;
	pTail	: POINTER TO ST_Pointer;
	pCurrent: POINTER TO ST_Pointer;
	nCount	: UINT;
END_VAR

METHOD M_Add
VAR_INPUT
	pStep : POINTER TO ST_Step;
END_VAR

VAR
	pNew : POINTER TO ST_Pointer;
END_VAR
//Checken, ob Step schon in Queue
pNew := pHead;
WHILE pNew > 0 DO
	IF pNew^.pContent = pStep THEN
		RETURN;
	END_IF
	pNew := pNew^.pNext;
END_WHILE

pNew := __NEW(ST_Pointer);
MEMSET(pNew,0,SIZEOF(ST_Pointer));
pNew^.pContent := pStep;
IF pHead = 0 THEN
	pHead := pTail := pNew;
ELSE
	pNew^.pPrev := pTail; 
	pTail^.pNext := pNew;
	pTail := pNew;
END_IF
nCount := nCount + 1;
END_METHOD

METHOD M_Get : POINTER TO ST_Step
VAR_INPUT
END_VAR

VAR
	pStep : POINTER TO ST_Step;
END_VAR
IF pCurrent > 0 THEN
	pStep := pCurrent^.pContent;
	IF pStep > 0 THEN
		IF pStep^.eState <> E_StepState.STEPSTATUS_Idle THEN
			M_Get := pStep;
		END_IF
	END_IF
	pCurrent := pCurrent^.pNext;
END_IF
END_METHOD

METHOD M_Remove : ERRORID
VAR_INPUT
	pStep : POINTER TO ST_STEP;
END_VAR

VAR
	pSeek : POINTER TO ST_Pointer;
	pTemp : POINTER TO ST_Pointer;
END_VAR
//Step in Queue suchen
pSeek := pHead;
WHILE pSeek > 0 DO
	IF pSeek^.pContent = pStep THEN
		//Anfang
		IF pSeek = pHead THEN	//Gesuchter ist Head
			IF pSeek^.pNext > 0 THEN //hat Nachfolger
				pHead := pSeek^.pNext;
				pHead^.pPrev := 0;
				//Wenn der zu löschende der aktuelle, dann wird der nächste der aktuelle
				IF pSeek = pCurrent THEN
					pCurrent := pHead^.pNext;
				END_IF
			ELSE //hat keinen Nachfolger
				pHead := 0;
				pTail := 0;
				pCurrent := 0;
			END_IF
		ELSIF pSeek = pTail THEN //Gesuchter ist Tail
			//Vorgänger wird Tail
			pTail := pTail^.pPrev;
			pTail^.pNext := 0;
			IF pSeek = pCurrent THEN
				pCurrent := 0;
			END_IF
 		ELSE //Gesuchter ist in der Mitte
			//Nachfolger beim Vorgänger eintragen
			pTemp := pSeek^.pPrev;
			pTemp^.pNext := pSeek^.pNext;
			//Vorganger beim Nachfolger eintragen
			pTemp := pSeek^.pNext;
			pTemp^.pPrev := pSeek^.pPrev;
			IF pSeek = pCurrent THEN
				pCurrent := pSeek^.pNext;
			END_IF
		END_IF
		__DELETE(pSeek);
		nCount := nCount - 1;
	ELSE
		pSeek := pSeek^.pNext;
	END_IF
END_WHILE
END_METHOD

METHOD M_Reset
VAR_INPUT
END_VAR

VAR
	pDelete : POINTER TO ST_Pointer;
	pNext	: POINTER TO ST_Pointer;
END_VAR
pDelete := pHead;
WHILE  pDelete > 0 DO
	pNext := pDelete^.pNext;
	__DELETE(pDelete);
	pDelete := pNext;
END_WHILE
pHead := 0;
pTail := 0;
pCurrent := 0;
nCount := 0;
END_METHOD

METHOD M_SetCurrentToHead
VAR_INPUT
END_VAR

VAR
	pStep : POINTER TO ST_Step;
END_VAR
pCurrent := pHead;
//Die Steps, die noch in "Idle" sind, in "InQueue" setzen
//Nur diese werden durch "M_Get" zurückgegeben
WHILE pCurrent > 0 DO
	pStep := pCurrent^.pContent;
	IF pStep^.eState = E_StepState.STEPSTATUS_Idle THEN
		pStep^.eState := E_StepState.STEPSTATUS_InQueue;
	END_IF
	pCurrent := pCurrent^.pNext;
END_WHILE
pCurrent := pHead;
END_METHOD

PROPERTY P_bEmpty : BOOL
GET
IF pHead = 0 AND pTail = 0 THEN
	P_bEmpty := TRUE;
END_IF
END_GET
END_PROPERTY

END_FUNCTION_BLOCK

// ---- Actions/ActionDispacher.TcPOU
PROGRAM ActionDispacher
VAR_OUTPUT
	eCurrentState 	: E_MachineState := E_MachineState.MACHINESTATE_Idle;
END_VAR
VAR
	stAction 			: ST_Action;
	pAction 			: POINTER TO ST_Action;
	nActionIdIntern		: UINT;
	fbActionList 		: FB_ActionList;
	fbDelayAction 		: FB_DelayAction;
	fbActionStatusList 	: FB_ActionStatusList;
	stActionStatus 		: ST_ActionStatus;	//für Notification
	eLastActionStatus	: E_ActionStatus;
	stError				: ST_Error;
	ppHElectrode		: POINTER TO FB_pHElectrode;
	
	bPauseRequestIntern	: BOOL;	//Flag für Sequence
	bLastActionResult	: BOOL;
	nLastActionResult	: DINT;	
	
	nStateA_Perform 	: USINT;
	nStateA_Reset 		: USINT;
	nStateA_StopAll 	: USINT;
	bErrorOnStopAll		: BOOL;
	bErrorOnReset		: BOOL;
	
	i					: UINT;
	
	nTest				: DINT;
	iDevice				: I_Device;
	iter				: FB_ObjCollectIterator;
END_VAR

CASE eCurrentState OF
	E_MachineState.MACHINESTATE_Idle:
		nStateA_Perform := 0;
		nStateA_StopAll := 0;
		nStateA_Reset := 0;
	E_MachineState.MACHINESTATE_Active:
		A_Perform();
		IF nStateA_Perform = 80 THEN
			eCurrentState := E_MachineState.MACHINESTATE_Idle;
		ELSIF nStateA_Perform = 99 THEN
			eCurrentState := E_MachineState.MACHINESTATE_Error;
		END_IF
	E_MachineState.MACHINESTATE_Cancel:
		A_StopAll();
		IF nStateA_StopAll = 80 THEN
			eCurrentState := E_MachineState.MACHINESTATE_Idle;
		ELSIF nStateA_StopAll = 99 THEN
 			eCurrentState := E_MachineState.MACHINESTATE_Error;
		END_IF
	E_MachineState.MACHINESTATE_Reset:
		A_Reset();
		IF nStateA_Reset = 80 THEN
			eCurrentState := E_MachineState.MACHINESTATE_Idle;
		ELSIF nStateA_Reset = 99 THEN
			eCurrentState := E_MachineState.MACHINESTATE_Error;
		END_IF
END_CASE

IF eCurrentState = E_MachineState.MACHINESTATE_Error THEN
	A_StopAll();
END_IF

//Actio status melden
fbActionStatusList.M_GetHead(stActionStatus);

//ActionList aufräumen
//eine Action bleibt noch einen Zyklus in der ActionList stehen, damit SequSteps sich noch
//den letzten Progresswert und den ActionResult holen können 
//Actions, welche welche in Ready oder Error sind werden gelöscht
//CleanUp
fbActionList.M_CleanUp();

ACTION A_Perform:
nStateA_Perform := 80;

fbActionList.M_SetCurrentToHead();
REPEAT
	pAction := fbActionList.M_GetNext();
	IF pAction > 0 THEN
		IF pAction^.eActionStatus >= E_ActionStatus.ACTIONSTATUS_Active AND pAction^.eActionStatus <= E_ActionStatus.ACTIONSTATUS_Pause THEN
			IF pAction^.eAction = E_Action.ACTION_Delay THEN //Delay
				fbDelayAction();
				pAction^.nProgress := fbDelayAction.M_GetProgress(UINT_TO_USINT(pAction^.stActionData.nObject));
				IF fbDelayAction.M_GetRestTime(UINT_TO_USINT(pAction^.stActionData.nObject)) = T#0S THEN
					//in nObject steht die TimerNr
					fbDelayAction.M_ReleaseTimer(UINT_TO_USINT(pAction^.stActionData.nObject));
					pAction^.eActionStatus := E_ActionStatus.ACTIONSTATUS_Ready;
				END_IF
			ELSIF pAction^.eAction = E_Action.ACTION_RunGCode THEN //GCode
				IF GCode.eGCodeState = E_GCodeState.GCodeState_Idle THEN
					pAction^.eActionStatus := E_ActionStatus.ACTIONSTATUS_Ready;
					pAction^.nProgress := 100;
				ELSIF GCode.eGCodeState = E_GCodeState.GCodeState_Running THEN
					pAction^.eActionStatus := E_ActionStatus.ACTIONSTATUS_Active;
					pAction^.nProgress := GCode.P_nProgress;
				ELSIF GCode.eGCodeState = E_GCodeState.GCodeState_Pause THEN
					pAction^.eActionStatus := E_ActionStatus.ACTIONSTATUS_Pause;
				ELSIF GCode.eGCodeState = E_GCodeState.GCodeState_ContinueRequest THEN
					pAction^.eActionStatus := E_ActionStatus.ACTIONSTATUS_Active;
				ELSIF GCode.eGCodeState = E_GCodeState.GCodeState_Error THEN
					pAction^.eActionStatus := E_ActionStatus.ACTIONSTATUS_Error;
					nStateA_Perform := 99;
				END_IF
			ELSIF pAction^.eAction = E_Action.ACTION_ShiftGCodeZPos THEN //GCode
				pAction^.eActionStatus := E_ActionStatus.ACTIONSTATUS_Ready;
			ELSIF pAction^.eAction = E_Action.ACTION_RunSequence THEN //Run Sequence
				pAction^.pSequence^();
				pAction^.nProgress := pAction^.pSequence^.P_nProgress;
				IF NOT pAction^.bExtern THEN
					nTest := pAction^.nProgress;
				END_IF
				IF (pAction^.pSequence^.eCurrentState = E_SequenceState.State_Ready OR
					pAction^.pSequence^.eCurrentState = E_SequenceState.State_Canceled) THEN
					pAction^.eActionStatus := E_ActionStatus.ACTIONSTATUS_Ready;
					//pAction^.nProgress := 100;
				ELSIF pAction^.pSequence^.eCurrentState = E_SequenceState.State_Pause THEN
					pAction^.eActionStatus := E_ActionStatus.ACTIONSTATUS_Pause;
				ELSIF pAction^.pSequence^.eCurrentState = E_SequenceState.State_Active THEN
					IF pAction^.eActionStatus <> E_ActionStatus.ACTIONSTATUS_Active THEN
						//tritt ein, wenn Sequenz in pause war -> ActionStatus wieder auf active setzen
						pAction^.eActionStatus := E_ActionStatus.ACTIONSTATUS_Active;
					END_IF
				ELSIF pAction^.pSequence^.eCurrentState = E_SequenceState.State_Error THEN
					pAction^.eActionStatus := E_ActionStatus.ACTIONSTATUS_Error;
					nStateA_Perform := 99;
				END_IF
			ELSIF pAction^.eAction = E_Action.ACTION_CoupleHeads THEN //Couple/Decouple YY-Axis (only platform d)
				CoupleYY();
				IF NOT CoupleYY.bBusy THEN
					IF CoupleYY.bError THEN
						pAction^.eActionStatus := E_ActionStatus.ACTIONSTATUS_Error;
						nStateA_Perform := 99;
					ELSE
						pAction^.eActionStatus := E_ActionStatus.ACTIONSTATUS_Ready;
					END_IF
					CoupleYY(bExecute:= FALSE);
				END_IF
			ELSIF pAction^.eAction >= 50 AND pAction^.eAction < 1000 THEN //BasicAction
				IF pAction^.iDevice.P_bError THEN
					stError := pAction^.iDevice.P_stError;
					pAction^.nErrorId := stError.ErrorId;
					pAction^.eActionStatus := E_ActionStatus.ACTIONSTATUS_Error;
					nStateA_Perform := 99;
				ELSE
					IF NOT pAction^.iDevice.M_GetActionBusy(eAction:= pAction^.eAction) THEN 
						IF pAction^.eAction = E_Action.ACTION_MeasurepH THEN
							ppHElectrode := pAction^.iDevice.P_pObject;
							bLastActionResult := TRUE;
							nLastActionResult := ppHElectrode^.P_nCurrentpHValue;
						END_IF
						pAction^.eActionStatus := E_ActionStatus.ACTIONSTATUS_Ready;
					END_IF
				END_IF
			ELSIF pAction^.eAction >= 1000 THEN	//ComplexAction
				IF NOT fbComplexAction.bBusy THEN
					bPauseRequestIntern := fbComplexAction.P_bPauseRequestIntern;
					fbComplexAction.P_bPauseRequestIntern := FALSE;
					IF fbComplexAction.bError THEN
						pAction^.eActionStatus := E_ActionStatus.ACTIONSTATUS_Error;
						nStateA_Perform := 99;
					ELSE
						IF fbComplexAction.P_bLastActionResult THEN
							bLastActionResult := TRUE;
							nLastActionResult := fbComplexAction.P_nLastActionResult;
							fbComplexAction.P_bLastActionResult := FALSE;
						END_IF
						pAction^.eActionStatus := E_ActionStatus.ACTIONSTATUS_Ready;
					END_IF
				ELSIF fbComplexAction.eCurrentState = E_MachineState.MACHINESTATE_PauseRequest THEN
					pAction^.eActionStatus := E_ActionStatus.ACTIONSTATUS_PauseRequest;
				ELSIF fbComplexAction.eCurrentState = E_MachineState.MACHINESTATE_Pause THEN
					pAction^.eActionStatus := E_ActionStatus.ACTIONSTATUS_Pause;
				ELSIF fbComplexAction.eCurrentState = E_MachineState.MACHINESTATE_Active THEN
					pAction^.eActionStatus := E_ActionStatus.ACTIONSTATUS_Active;
				END_IF	
			END_IF
			fbActionStatusList.M_AddTail(pAction);
		END_IF			
	END_IF

UNTIL pAction = 0
END_REPEAT

IF nStateA_Perform = 80 THEN
	IF fbActionList.P_bActionsAvailable THEN
		nStateA_Perform := 0;
	END_IF
END_IF
END_ACTION

ACTION A_Reset:
IF nStateA_Reset = 0 THEN
	bErrorOnReset := FALSE;
	fbObjectDirectory.P_pDeviceCollection^.M_GetIterator(iter);
	WHILE iter.pNode > 0 AND_THEN iter.pNode^.P_pObject > 0 DO
		iDevice := iter.pNode^.P_pObject^.M_GetDevice();
		IF iDevice <> 0 THEN
			IF iDevice.P_bError THEN
				iDevice.M_Reset();
			ELSIF iDevice.P_bBusy THEN
				iDevice.M_Stop();
			END_IF
		END_IF
		iter.M_Increment();
	END_WHILE
	
	IF fbComplexAction.bError THEN	//Die ResetMethode von fbComplexAction 1x aufrufen 
		fbComplexAction.M_Reset();	
	END_IF
	
	IF GCode.bError THEN
		GCode.M_Reset();
	END_IF

	fbSequenceList.M_ResetAllSequ();
	
	nStateA_Reset := 1;
	
ELSIF nStateA_Reset = 1 THEN
	nStateA_Reset := 2;
	fbObjectDirectory.P_pDeviceCollection^.M_GetIterator(iter);
	WHILE iter.pNode > 0 AND_THEN iter.pNode^.P_pObject > 0 DO
		iDevice := iter.pNode^.P_pObject^.M_GetDevice();
		IF iDevice <> 0 THEN
			IF NOT iDevice.P_bBusy THEN
				IF iDevice.P_bError THEN
					bErrorOnReset := TRUE;
				END_IF
			ELSE
				nStateA_Reset := 1;
			END_IF
		END_IF
		iter.M_Increment();
	END_WHILE
	
	
	IF NOT fbComplexAction.bBusy THEN
		IF fbComplexAction.bError THEN
			bErrorOnReset := TRUE;
		END_IF
	ELSE
		nStateA_Reset := 1;
	END_IF
	
ELSIF nStateA_Reset = 2 THEN
	IF bErrorOnReset THEN
		nStateA_Reset := 99;
	ELSE
		nStateA_Reset := 80;
	END_IF
END_IF
END_ACTION

ACTION A_StopAll:
IF nStateA_StopAll = 0 THEN
	bErrorOnStopAll := FALSE;
	//Nur externe Actions stoppen
	fbActionList.M_SetCurrentToHead();
	REPEAT
		pAction := fbActionList.M_GetNext();
		IF pAction > 0 THEN
			IF pAction^.bExtern AND pAction^.eActionStatus >= E_ActionStatus.ACTIONSTATUS_Active AND
										pAction^.eActionStatus <= E_ActionStatus.ACTIONSTATUS_Pause THEN
				M_StopAction(pAction^.nActionId);	
			END_IF
		END_IF
	UNTIL pAction = 0
	END_REPEAT
	nStateA_StopAll := 1;
ELSIF nStateA_StopAll = 1 THEN	//alle Actions gestoppt?
	nStateA_StopAll := 2;
	fbActionList.M_SetCurrentToHead();
	REPEAT
		pAction := fbActionList.M_GetNext();
		IF pAction > 0 THEN
			IF pAction^.eActionStatus >= E_ActionStatus.ACTIONSTATUS_Active AND pAction^.eActionStatus <= E_ActionStatus.ACTIONSTATUS_Pause THEN
				IF pAction^.eAction = E_Action.ACTION_Delay THEN
					fbDelayAction();
					IF fbDelayAction.M_GetRestTime(UINT_TO_USINT(pAction^.stActionData.nObject)) = T#0S THEN
						pAction^.eActionStatus := E_ActionStatus.ACTIONSTATUS_Ready;
					END_IF
				ELSIF pAction^.eAction = E_Action.ACTION_RunGCode THEN //GCode
					IF GCode.eGCodeState = E_GCodeState.GCodeState_Idle THEN
						pAction^.eActionStatus := E_ActionStatus.ACTIONSTATUS_Ready;
					ELSIF GCode.eGCodeState = E_GCodeState.GCodeState_Error THEN
						pAction^.eActionStatus := E_ActionStatus.ACTIONSTATUS_Error;
					END_IF
				ELSIF pAction^.eAction = E_Action.ACTION_RunSequence THEN //Run Sequence
					pAction^.pSequence^();
					IF (pAction^.pSequence^.eCurrentState = E_SequenceState.State_Ready OR
						pAction^.pSequence^.eCurrentState = E_SequenceState.State_Canceled) THEN
						pAction^.eActionStatus := E_ActionStatus.ACTIONSTATUS_Ready;
					ELSIF pAction^.pSequence^.eCurrentState = E_SequenceState.State_Error THEN
						pAction^.eActionStatus := E_ActionStatus.ACTIONSTATUS_Error;
					END_IF
				ELSIF pAction^.eAction >= 50 AND pAction^.eAction < 1000 THEN //BasicAction
					IF pAction^.iDevice.P_bError THEN
						pAction^.eActionStatus := E_ActionStatus.ACTIONSTATUS_Error;
					ELSE
						IF NOT pAction^.iDevice.M_GetActionBusy(eAction:= pAction^.eAction) THEN 
							pAction^.eActionStatus := E_ActionStatus.ACTIONSTATUS_Ready;
						END_IF
					END_IF
				ELSIF pAction^.eAction >= 1000 THEN	//ComplexAction
					IF NOT fbComplexAction.bBusy THEN
						IF fbComplexAction.bError THEN
							pAction^.eActionStatus := E_ActionStatus.ACTIONSTATUS_Error;
						ELSE
							pAction^.eActionStatus := E_ActionStatus.ACTIONSTATUS_Ready;
						END_IF
					END_IF	
				END_IF
				
				fbActionStatusList.M_AddTail(pAction);
				
				IF pAction^.eActionStatus = E_ActionStatus.ACTIONSTATUS_Ready THEN
					;//do nothing
				ELSIF pAction^.eActionStatus = E_ActionStatus.ACTIONSTATUS_Error THEN
					bErrorOnStopAll := TRUE;
				ELSE
					nStateA_StopAll := 1;
				END_IF
			END_IF
		END_IF
	UNTIL pAction = 0
	END_REPEAT
ELSIF nStateA_StopAll = 2 THEN
	//Bei allen Devices, die Busy sind, die Stop-Methode aufrufen
	
	(*IF fbObjectDirectory.nCntDevice > 0 THEN
		FOR i:= 1 TO fbObjectDirectory.nCntDevice BY 1 DO
			IF aI_Device[i].P_bBusy THEN	//Devices die noch Busy sind, stoppen
				aI_Device[i].M_Stop();
			END_IF;
			IF aI_Device[i].P_bError THEN
				bErrorOnStopAll := TRUE;
			END_IF
		END_FOR
	END_IF*)		
	IF bErrorOnStopAll THEN
		nStateA_StopAll := 99;
	ELSE
		nStateA_StopAll := 80;
	END_IF
END_IF
END_ACTION

METHOD M_ContinueAction : ERRORID
VAR_INPUT
	nActionId : UINT;
END_VAR

VAR_OUTPUT
	nProgress	: UINT;
END_VAR

VAR
	pAction : POINTER TO ST_Action;
END_VAR
pAction := fbActionList.M_GetFromId(nActionId);
IF pAction > 0 THEN
	IF pAction^.eActionStatus = E_ActionStatus.ACTIONSTATUS_Pause THEN
		IF pAction^.eAction = E_Action.ACTION_RunGCode THEN
			GCode.M_Continue();
			nProgress := GCode.P_nProgress;
			RETURN;
		ELSIF pAction^.eAction = E_Action.ACTION_RunSequence THEN
			pAction^.pSequence^.M_Continue();
			RETURN;
		ELSIF pAction^.eAction = E_Action.ACTION_DispenseTest THEN
			fbComplexAction.M_Continue();
			RETURN;
		ELSIF pAction^.eAction = E_Action.ACTION_Delay THEN
			pAction^.eActionStatus := E_ActionStatus.ACTIONSTATUS_Active;
			RETURN;
		END_IF
	END_IF
END_IF
M_ContinueAction := E_ErrorIdCmd.ERRORID_InvalidAction;
END_METHOD

METHOD M_ExeAction : ERRORID
VAR_INPUT
	refActionData	: REFERENCE TO ST_ActionData;
	bExtern			: BOOL;	
END_VAR
VAR_OUTPUT
	nActionId		: UINT;
END_VAR
VAR
	nObjectId			: UINT;
	iDevice				: I_Device;
	pSequence			: POINTER TO FB_Sequence;
	sGCodeFileNumber	: STRING;
	i					: UINT;
	
END_VAR
//Actions werden nur in Idle, Active und Ready entgegengenommen
//erfolgreich angenommene Actions liefern eine Id zurück, welche die Action eindeutig identifiziert
//anhand dieser Id kann über die Methode "M_GetActionStatus(nActionId)" festgestellt werden, ob Action fertig
IF NOT ((eCurrentState = E_MachineState.MACHINESTATE_Idle) OR (eCurrentState = E_MachineState.MACHINESTATE_Active)) THEN
	M_ExeAction := E_ErrorIdCmd.ERRORID_InvalidState;
	RETURN;
END_IF

iDevice := 0;
stAction.pSequence := 0;

//Unterscheidung zwischen GCode-Control-Actions, BasicActions, ComplexActions und DelayAction

//Erste Unterscheidung zwischen ControlActions, BasicActions und ComplexActions
IF refActionData.eAction > 0 AND refActionData.eAction < 50 THEN //ControlActions
	CASE refActionData.eAction OF
		E_Action.ACTION_Delay:
			refActionData.nObject := fbDelayAction.M_StartTimer(DINT_TO_TIME(refActionData.aParams[1]));
			IF refActionData.nObject = 0 THEN
				//in nObject steht die TimerNr
				M_ExeAction := E_ErrorIdCmd.ERRORID_NoFreeTimerAvailable;
				RETURN;
			END_IF
		E_Action.ACTION_GoToStep:
			RETURN;
		E_Action.ACTION_RunGCode:
			IF NOT GCode.P_bNciAvailable THEN
				M_ExeAction := E_ErrorIdGCode.ERRORID_NciModuleNotAvailable;
				RETURN;	
			END_IF	
			//Nur ausführbar, wenn GCode-Modul noch nicht läuft
			IF GCode.eGCodeState = E_GCodeState.GCodeState_Idle THEN
				//Startnullpunkt setzen
				M_ExeAction := GCode.M_SetStartZeroPoint(refActionData.nTarget,
										DINT_TO_USINT(refActionData.aParams[1]),
										DINT_TO_UINT(refActionData.aParams[2]),
										DINT_TO_UINT(refActionData.aParams[3]),
										refActionData.aParams[4],
										DINT_TO_UINT(refActionData.aParams[6]),
										DINT_TO_REAL(refActionData.aParams[7]),
										DINT_TO_USINT(refActionData.aParams[8]));
				IF M_ExeAction > 0 THEN
					RETURN;
				END_IF
				//übergebene SequenceIds checken
				FOR i := 9 TO 13 BY 1 DO
					IF refActionData.aParams[i] > 0 THEN
						IF fbSequenceList.M_Get(DINT_TO_UDINT(refActionData.aParams[i])) = 0 THEN
							M_ExeAction := E_ErrorIdCmd.ERRORID_SequenceNotExists;
							RETURN;
						END_IF
					END_IF
				END_FOR
				GCode.M_SetSequenceIds(ADR(refActionData.aParams[9]));
				
				sGCodeFileNumber := DINT_TO_STRING(refActionData.aParams[5]);
				GCode.M_Start(sGCodeFileNumber);
			ELSE
				M_ExeAction := E_ErrorIdGCode.ERRORID_InvalidNciState;
				RETURN;
			END_IF
		
		E_Action.ACTION_ShiftGCodeZPos:
			IF NOT GCode.P_bNciAvailable THEN
				M_ExeAction := E_ErrorIdGCode.ERRORID_NciModuleNotAvailable;
				RETURN;	
			END_IF	
			GCode.M_ShiftZPos(DINT_TO_REAL(refActionData.aParams[1]));
		
		E_Action.ACTION_RunSequence:
			pSequence := fbSequenceList.M_Get(DINT_TO_UDINT(refActionData.aParams[1]));
			IF pSequence > 0 THEN
				//Sequence muss im Idle sein
				M_ExeAction := pSequence^.M_CheckForStart();
				IF M_ExeAction > 0 THEN
					RETURN;
				ELSE
					//refActionData.aParams[2] nur für Aufruf von SubSequences aus MainSequence wenn
					//in der SubSequence ein MoveToTarget mit TargetRef "SequParaToArrayItem" benutzt wird
					//Somit kann auf einem Array eine SubSequence ausgeführt werden
					pSequence^.M_Start(DINT_TO_UINT(refActionData.aParams[2]));
					stAction.pSequence := pSequence;
				END_IF
			ELSE
				//Sequence mit angegebener Id nicht vorhanden
				M_ExeAction := E_ErrorIdCmd.ERRORID_SequenceNotExists;
				RETURN;							
			END_IF
		E_Action.ACTION_CoupleHeads:
			(*Die erste Ausführung des KoppelBausteins erfolgt bereits hier, so kann bei einer ungültigen
			Startbedingung hier schon der Abbruch erfolgen*)
			CoupleYY(bCouple:= DINT_TO_BOOL(refActionData.aParams[1]),bExecute:= TRUE,nErrorID=> M_ExeAction);
			IF CoupleYY.bError THEN
				CoupleYY(bExecute:= FALSE);
				RETURN;
			END_IF
	END_CASE

ELSIF refActionData.eAction >= 50 AND refActionData.eAction < 1000 THEN //BasicActions
	//Nur ausführbar, wenn GCode-Modul MoveActions nicht sperrt
	IF GCode.P_bMoveActionsLocked AND_THEN (refActionData.eAction = E_Action.ACTION_MoveX OR
				 							refActionData.eAction = E_Action.ACTION_MoveY OR
				 							refActionData.eAction = E_Action.ACTION_MoveZ OR
				 							refActionData.eAction = E_Action.ACTION_MoveXY) THEN
		//Action nicht ausführbar, da von GCodeModul gesperrt
		M_ExeAction := E_ErrorIdCmd.ERRORID_ActionLocked;
		RETURN;
	END_IF
	nObjectId := refActionData.nObject;
	//Gültiges Device?
	IF NOT fbObjectDirectory.M_ObjIsDevice(nObjectId) THEN
		M_ExeAction := E_ErrorIdObjMgmt.ERRORID_IsNoDevice;	//Error: Object ist kein Device
		RETURN;
	END_IF
	iDevice := fbObjectDirectory.M_GetDevice(nObjectId);
	M_ExeAction := iDevice.M_ExeAction(refActionData);	//Action an Device ausführen
	IF 	M_ExeAction > 0 THEN
		RETURN;
	END_IF
ELSE //ComplexActions
	//Nur ausführbar, wenn GCode-Modul MoveActions nicht sperrt
	IF GCode.P_bMoveActionsLocked THEN
		M_ExeAction := E_ErrorIdCmd.ERRORID_ActionLocked;
		RETURN;
	END_IF
	
	M_ExeAction := fbComplexAction.M_ExeAction(refActionData);	//ComplexeAction ausführen
	IF 	M_ExeAction > 0 THEN
		RETURN;
	END_IF
END_IF

//Neue ActionId bilden
//darf nicht bereits durch aktive Action belegt sein
//das kann vorkommen, wenn es einen Überlauf gibt bei Sequenzen mit > 65535 Steps
nActionIdIntern := nActionIdIntern + 1;
WHILE fbActionList.M_GetFromId(nActionIdIntern) > 0 DO
	nActionIdIntern := nActionIdIntern + 1;
END_WHILE
nActionId := nActionIdIntern;
stAction.nActionId := nActionId;
stAction.eAction := refActionData.eAction;
stAction.iDevice := iDevice;
stAction.stActionData := refActionData;
stAction.eActionStatus := E_ActionStatus.ACTIONSTATUS_Active;
stAction.eActionStatusOld := E_ActionStatus.ACTIONSTATUS_Idle;
stAction.nErrorId := 0;
stAction.bExtern := bExtern;

fbActionList.M_Add(stAction);
fbActionStatusList.M_AddTail(ADR(stAction));
eCurrentState := E_MachineState.MACHINESTATE_Active;
END_METHOD

METHOD M_GetActionInfoArray
VAR_INPUT
	pActiveActionArray : POINTER TO ARRAY[0..0] OF ST_ActionStatus;
END_VAR

VAR
	pAction : POINTER TO ST_Action;
	i 		: USINT;
END_VAR
MEMSET(pActiveActionArray,0,90);
fbActionList.M_SetCurrentToHead();
REPEAT
	pAction := fbActionList.M_GetNext();
	IF pAction > 0 THEN
		IF pAction^.bExtern THEN
			pActiveActionArray^[i].nActionId := pAction^.nActionId;
			pActiveActionArray^[i].eAction := pAction^.eAction;
			pActiveActionArray^[i].eStatus := pAction^.eActionStatus;
			pActiveActionArray^[i].nObjectId := pAction^.stActionData.nObject;
			//MultiChannelActions
			IF pAction^.eAction = E_Action.ACTION_SetPressure OR pAction^.eAction = E_Action.ACTION_SwitchPressure THEN
				pActiveActionArray^[i].nChannel := DINT_TO_USINT(pAction^.stActionData.aParams[1]);
			END_IF			
			i := i + 1;
		END_IF
	END_IF
UNTIL (pAction = 0) OR (i = 9)
END_REPEAT
END_METHOD

METHOD M_GetActionStatus : E_ActionStatus
VAR_INPUT
	nActionId	: UINT;
END_VAR

VAR_OUTPUT
	nProgress	: UINT;	
END_VAR

VAR
	pAction : POINTER TO ST_Action;
END_VAR
pAction := fbActionList.M_GetFromId(nActionId);
IF pAction > 0 THEN
	nProgress := pAction^.nProgress;
	M_GetActionStatus := pAction^.eActionStatus;
	RETURN;
END_IF
M_GetActionStatus := E_ActionStatus.ACTIONSTATUS_Ready;
END_METHOD

METHOD M_PauseAction : ERRORID
VAR_INPUT
	nActionId : UINT;
END_VAR

VAR
	pAction : POINTER TO ST_Action;
END_VAR
pAction := fbActionList.M_GetFromId(nActionId);
IF pAction > 0 THEN
	IF pAction^.eActionStatus = E_ActionStatus.ACTIONSTATUS_Active THEN
		IF pAction^.eAction = E_Action.ACTION_RunGCode THEN
			GCode.M_Pause();
			RETURN;
		ELSIF pAction^.eAction = E_Action.ACTION_RunSequence THEN
			pAction^.pSequence^.M_Pause();
			RETURN;
		ELSIF pAction^.eAction = E_Action.ACTION_DispenseTest THEN
			fbComplexAction.M_Pause();
			RETURN;
		ELSIF pAction^.eAction = E_Action.ACTION_Delay THEN
			pAction^.eActionStatus := E_ActionStatus.ACTIONSTATUS_Pause;
		END_IF				
	END_IF
END_IF
M_PauseAction := E_ErrorIdCmd.ERRORID_InvalidAction;
END_METHOD

METHOD M_Reset
VAR_INPUT
END_VAR
IF eCurrentState = E_MachineState.MACHINESTATE_Error THEN
	eCurrentState := E_MachineState.MACHINESTATE_Reset;
END_IF;
END_METHOD

METHOD M_StopAction : ERRORID
VAR_INPUT
	nActionId : UINT;
END_VAR

VAR
	pAction : POINTER TO ST_Action;
END_VAR
pAction := fbActionList.M_GetFromId(nActionId);
IF pAction > 0 THEN
	IF pAction^.eAction = E_Action.ACTION_Delay THEN
		//Delay abbrechen
		fbDelayAction.M_ReleaseTimer(UINT_TO_USINT(pAction^.stActionData.nObject));
	ELSIF pAction^.eAction = E_Action.ACTION_RunSequence THEN
		pAction^.pSequence^.M_Stop();
		RETURN;
	ELSIF pAction^.eAction = E_Action.ACTION_RunGCode THEN
		IF NOT GCode.P_bNciAvailable THEN
			M_StopAction := E_ErrorIdGCode.ERRORID_NciModuleNotAvailable;
			RETURN;
		END_IF	
		//Nur ausführbar, wenn GCode-Modul in Pause oder Running
		//wird nicht in ActionList eingetragen
		IF GCode.eGCodeState <> E_GCodeState.GCodeState_Idle THEN
			GCode.M_Stop();
			RETURN;
		ELSE
			M_StopAction := E_ErrorIdGCode.ERRORID_InvalidNciState;
		END_IF
	ELSIF pAction^.eAction >= 50 AND pAction^.eAction < 1000 THEN
		pAction^.iDevice.M_CancelAction(pAction^.eAction);
		RETURN;
	ELSIF pAction^.eAction >= 1000 THEN
		fbComplexAction.M_StopAction(pAction^.eAction);
		RETURN;
	ELSIF pAction^.eAction = E_Action.ACTION_Delay THEN
		fbDelayAction.M_ReleaseAll();
		RETURN;
	END_IF			
END_IF
M_StopAction := E_ErrorIdCmd.ERRORID_InvalidAction;
END_METHOD

METHOD M_StopAll
VAR_INPUT
END_VAR
IF eCurrentState = E_MachineState.MACHINESTATE_Active THEN
	eCurrentState := E_MachineState.MACHINESTATE_Cancel;
END_IF
END_METHOD

PROPERTY P_bLastActionResult : BOOL
GET
P_bLastActionResult := bLastActionResult;
END_GET
SET
bLastActionResult := P_bLastActionResult;
fbComplexAction.P_bLastActionResult := bLastActionResult;
END_SET
END_PROPERTY

PROPERTY P_bPauseRequestIntern : BOOL
GET
P_bPauseRequestIntern := bPauseRequestIntern;
END_GET
SET
bPauseRequestIntern := P_bPauseRequestIntern;
fbComplexAction.P_bPauseRequestIntern := bPauseRequestIntern;
END_SET
END_PROPERTY

PROPERTY P_nActiveActions : UDINT
GET
P_nActiveActions := fbActionList.nCount;
END_GET
END_PROPERTY

PROPERTY P_nLastActionResult : DINT
GET
P_nLastActionResult := nLastActionResult;
END_GET
SET
nLastActionResult := P_nLastActionResult;
END_SET
END_PROPERTY

END_PROGRAM

// ---- Actions/FB_ActionList.TcPOU
FUNCTION_BLOCK FB_ActionList
VAR_INPUT
END_VAR
VAR_OUTPUT
END_VAR
VAR
	pHead	: POINTER TO ST_Pointer;
	pTail	: POINTER TO ST_Pointer;
	pCurrent: POINTER TO ST_Pointer;
	nCount	: UINT;
	pAction : POINTER TO ST_Action;
END_VAR

METHOD M_Add
VAR_INPUT
	stAction : REFERENCE TO ST_Action;
END_VAR

VAR
	pNew : POINTER TO ST_Pointer;
	pAction : POINTER TO ST_Action;
END_VAR
pNew := pHead;
WHILE pNew > 0 DO
	pAction := pNew^.pContent;
	//Action für das Device schon in Liste? Es sei denn, die Action ist bereits schon in Idle versetzt.
	IF (pAction^.eAction >= 50) AND (pAction^.iDevice = stAction.iDevice) AND (pAction^.eAction = stAction.eAction) AND pAction^.eActionStatus <> E_ActionStatus.ACTIONSTATUS_Idle THEN
		RETURN;
	END_IF
	pNew := pNew^.pNext;
END_WHILE

pNew := __NEW(ST_Pointer);
MEMSET(pNew,0,SIZEOF(ST_Pointer));
pAction := __NEW(ST_Action);
MEMCPY(pAction,ADR(stAction),SIZEOF(stAction));
pNew^.pContent := pAction;
IF pHead = 0 THEN
	pHead := pTail := pNew;
ELSE
	pNew^.pPrev := pTail; 
	pTail^.pNext := pNew;
	pTail := pNew;
END_IF
nCount := nCount + 1;
END_METHOD

METHOD M_CleanUp
VAR_INPUT
END_VAR
VAR
	pSeek : POINTER TO ST_Pointer;
	pTemp : POINTER TO ST_Pointer;
	pAction : POINTER TO ST_Action;
END_VAR
//Actions, welche Ready oder in Error gegangen sind in Idle setzen (werden beim nächsten Aufruf gelöscht)
pSeek := pHead;
WHILE (pSeek > 0) DO
	pAction := pSeek^.pContent;
	IF pAction^.eActionStatus = E_ActionStatus.ACTIONSTATUS_Ready OR pAction^.eActionStatus = E_ActionStatus.ACTIONSTATUS_Error THEN
		pAction^.eActionStatus := E_ActionStatus.ACTIONSTATUS_Idle;
		pSeek := pSeek^.pNext;
	ELSIF pAction^.eActionStatus = E_ActionStatus.ACTIONSTATUS_Idle THEN
		IF pSeek = pHead THEN	//Gesuchter ist Head
			IF pSeek^.pNext > 0 THEN //hat Nachfolger
				//Nachfolger wird zum Head
				pHead := pSeek^.pNext;
				pHead^.pPrev := 0; //Head hat keinen Vorgänger
				IF pSeek = pCurrent THEN
					pCurrent := 0;
				END_IF
			ELSE //hat keinen Nachfolger
				pHead := 0;
				pTail := 0;
				pCurrent := 0;				
			END_IF
		ELSIF pSeek = pTail THEN //pSeek ist Tail
			//Vorgänger wird Tail
			pTail := pTail^.pPrev;
			pTail^.pNext := 0; //Tail hat keinen Nachfolger
			IF pSeek = pCurrent THEN
				pCurrent := 0;
			END_IF
		ELSE //pSeek ist in der Mitte
			//Vorgänger beim Nachfolger eintragen
			pTemp := pSeek^.pPrev;
			pTemp^.pNext := pSeek^.pNext;
			//Vorganger beim Nachfolger eintragen
			pTemp := pSeek^.pNext;
			pTemp^.pPrev := pSeek^.pPrev;
			IF pSeek = pCurrent THEN
				pCurrent := pSeek^.pNext;
			END_IF			
		END_IF
		pTemp := pSeek;
		pSeek := pSeek^.pNext;
		__DELETE(pTemp);
		__DELETE(pAction);
		nCount := nCount - 1;		
	ELSE
		pSeek := pSeek^.pNext;
	END_IF
END_WHILE
END_METHOD

METHOD M_GetFromId : POINTER TO ST_Action
VAR_INPUT
	nActionId : UINT;
END_VAR

VAR
	pTemp : POINTER TO ST_Pointer;
	pAction : POINTER TO ST_Action;
END_VAR
pTemp := pHead;
WHILE (pTemp > 0) DO
	pAction := pTemp^.pContent;
	IF pAction^.nActionId = nActionId THEN
		M_GetFromId := pAction;
		RETURN;
	ELSE
		pTemp := pTemp^.pNext;
	END_IF
END_WHILE
END_METHOD

METHOD M_GetNext : POINTER TO ST_Action
VAR_INPUT
END_VAR
IF pCurrent > 0 THEN
	M_GetNext := pCurrent^.pContent;
	pCurrent := pCurrent^.pNext;
END_IF
END_METHOD

METHOD M_Reset
VAR_INPUT
END_VAR

VAR
	pDelete : POINTER TO ST_Pointer;
	pNext	: POINTER TO ST_Pointer;
	pAction : POINTER TO ST_Action;
END_VAR
pDelete := pHead;
WHILE  pDelete > 0 DO
	pAction := pDelete^.pContent;
	pNext := pDelete^.pNext;
	__DELETE(pAction);
	__DELETE(pDelete);
	pDelete := pNext;
END_WHILE
pHead := 0;
pTail := 0;
pCurrent := 0;
nCount := 0;
END_METHOD

METHOD M_SetCurrentToHead
VAR_INPUT
END_VAR
pCurrent := pHead;
END_METHOD

PROPERTY P_bActionsAvailable : BOOL
GET
VAR
	pTemp : POINTER TO ST_Pointer;
	pAction : POINTER TO ST_Action;
END_VAR
//Actions vorhanden die in Active, Pause oder Pause Request sind ?
pTemp := pHead;
WHILE (pTemp > 0) DO
	pAction := pTemp^.pContent;
	IF pAction^.eActionStatus >= E_ActionStatus.ACTIONSTATUS_Active AND pAction^.eActionStatus <= E_ActionStatus.ACTIONSTATUS_Pause THEN
		P_bActionsAvailable := TRUE;
		RETURN;
	ELSE
		pTemp := pTemp^.pNext;
	END_IF
END_WHILE
END_GET
END_PROPERTY

END_FUNCTION_BLOCK

// ---- Actions/FB_DelayAction.TcPOU
FUNCTION_BLOCK FB_DelayAction
VAR_INPUT
END_VAR
VAR_OUTPUT
END_VAR
VAR
	aTimer 		: ARRAY[1..cNoOfTimers] OF TON;
	nTimerNr 	: USINT; 
END_VAR

VAR CONSTANT
	cNoOfTimers : USINT := 4;
END_VAR

FOR nTimerNr := 1 TO cNoOfTimers BY 1 DO
	aTimer[nTimerNr]();
END_FOR

METHOD M_GetProgress : USINT
VAR_INPUT
	nTimerNr	: USINT;
END_VAR

VAR
	nPT : UDINT;
	nET : UDINT;
END_VAR
nPT := TIME_TO_UDINT(aTimer[nTimerNr].PT);
nET := TIME_TO_UDINT(aTimer[nTimerNr].ET);
M_GetProgress := UDINT_TO_USINT(nET * 100 / nPT);
END_METHOD

METHOD M_GetRestTime : TIME
VAR_INPUT
	nTimerNr	: USINT;
END_VAR
IF aTimer[nTimerNr].IN THEN
	M_GetRestTime := aTimer[nTimerNr].PT - aTimer[nTimerNr].ET;
END_IF
END_METHOD

METHOD M_ReleaseAll
VAR_INPUT
END_VAR
FOR nTimerNr := 1 TO cNoOfTimers BY 1 DO
	aTimer[nTimerNr](IN:= FALSE);
END_FOR
END_METHOD

METHOD M_ReleaseTimer
VAR_INPUT
	nTimerNr	: USINT;
END_VAR
aTimer[nTimerNr](IN:= FALSE);
END_METHOD

METHOD M_StartTimer : USINT
VAR_INPUT
	tTime	: TIME;
END_VAR
//nächsten freien Timer suchen
FOR nTimerNr := 1 TO cNoOfTimers BY 1 DO
	IF aTimer[nTimerNr].IN = FALSE THEN
		aTimer[nTimerNr](IN:= TRUE, PT:= tTime);
		M_StartTimer := nTimerNr;
		EXIT;
	END_IF
END_FOR
END_METHOD

END_FUNCTION_BLOCK

// ---- Actions/FB_ActionStatusList.TcPOU
FUNCTION_BLOCK FB_ActionStatusList
VAR_INPUT
END_VAR
VAR_OUTPUT
END_VAR
VAR
	pHead : POINTER TO ST_Pointer;
	pTail : POINTER TO ST_Pointer;
END_VAR

METHOD M_AddTail
VAR_INPUT
	pAction : POINTER TO ST_Action;
END_VAR

VAR
	pNewPointer : POINTER TO ST_Pointer;
	pNewContent : POINTER TO ST_ActionStatus;
END_VAR
//Es werden nur externe Actions in diese Liste aufgenommen,
//da diese auch nur zur GUI gemeldet werden müssen
IF pAction > 0 THEN
	IF pAction^.bExtern AND (pAction^.eActionStatus <> pAction^.eActionStatusOld) THEN
		pAction^.eActionStatusOld := pAction^.eActionStatus;
		pNewPointer := __NEW(ST_Pointer);
		pNewContent := __NEW(ST_ActionStatus);
		MEMSET(pNewPointer,0,SIZEOF(ST_Pointer));
		
		pNewContent^.nActionId := pAction^.nActionId;
		pNewContent^.eAction := pAction^.eAction;
		pNewContent^.eStatus := pAction^.eActionStatus;
		pNewContent^.nObjectId := pAction^.stActionData.nObject;
		
		pNewPointer^.pContent := pNewContent;
		
		IF pTail = 0 THEN
			pHead := pTail := pNewPointer;
		ELSE
			pNewPointer^.pPrev := pTail;
			pTail^.pNext := pNewPointer;
			pTail := pNewPointer;
		END_IF
	END_IF
END_IF
END_METHOD

METHOD M_GetHead
VAR_INPUT
END_VAR
VAR_IN_OUT
	stActionStatus : ST_ActionStatus;
END_VAR

VAR
	pContent	: POINTER TO ST_ActionStatus;
	pTemp		: POINTER TO ST_Pointer;
END_VAR
//Immer vom Head holen und dann löschen
IF pHead > 0 THEN
	MEMCPY(ADR(stActionStatus),pHead^.pContent,SIZEOF(stActionStatus));
	__DELETE(pHead^.pContent);
	IF pHead^.pNext > 0 THEN //Next wird zu Head
		pTemp := pHead^.pNext;
		__DELETE(pHead);
		pTemp^.pPrev := 0;
		pHead := pTemp;
	ELSE
		__DELETE(pHead);
		pTail := 0;
	END_IF
END_IF
END_METHOD

END_FUNCTION_BLOCK

// ---- Objects/Tools/FB_pHElectrode.TcPOU
FUNCTION_BLOCK FB_pHElectrode EXTENDS FB_MzTool
VAR_INPUT
END_VAR
VAR_OUTPUT
END_VAR
VAR
	//Specproperties
	nDigiOutChannelMz	: USINT;	//24V-Versorung für Messwertverstärker
	nAnaInputChannelMz	: USINT;	//Messwert (0-5V entsprechen pH0-14)
	
	pFbGPInputRef			: POINTER TO FB_GPInputRef;
	
	//****************************************Aktionvariablen****************************************************
	stActionDataSpec	: ST_ActionData;
	
	//Action: "InitTool"
	bInitTool			: BOOL;
	nStateA_InitTool	: USINT;
	
	//"Measure pH"
	bMeasurepH : BOOL;
	nStateA_MeasurepH : USINT;
	tTime 	: TIME;
	timer	: TON;
	
	
	rCurrentpHValue	: REAL;
END_VAR

IF eCurrentState = E_MachineState.MACHINESTATE_Active THEN
	IF bInitTool THEN
		A_InitTool();
		IF nStateA_InitTool >= 80 THEN
			IF nStateA_InitTool >= 99 THEN
				bError := TRUE;		
			END_IF
			bInitTool := FALSE;
			nStateA_InitTool := 0;
			M_RemoveListEntry(nSearchValue:= E_Action.ACTION_Init);
		END_IF		
	END_IF
	
	IF bMeasurepH THEN
		A_MeasurepH();
		IF nStateA_MeasurepH >= 80 THEN
			IF nStateA_MeasurepH >= 99 THEN
				bError := TRUE;
			END_IF
			bMeasurepH := FALSE;
			nStateA_MeasurepH := 0;
			M_RemoveListEntry(nSearchValue:= E_Action.ACTION_MeasurepH);
		END_IF
	END_IF

END_IF

//FB_MzTool aufrufen
SUPER^();

//Prozessdaten aktualisieren
IF pFbGPInputRef > 0 THEN
	rCurrentpHValue := 14.0 / 65535.0 * pFbGPInputRef^.nValue;
END_IF
stProcessData.n32Data[7] := REAL_TO_DINT(rCurrentpHValue * 1000.0);

aObjProcData[nNotifyId] := stProcessData;

ACTION A_InitTool:
IF nStateA_InitTool = 0 THEN
	pFbMultiZ^.aDigiOut[nDigiOutChannelMz] := TRUE;
	pFbGPInputRef^(eMode:= E_GPInputMode.Analog, bInit:= TRUE);
	IF NOT pFbGPInputRef^.bBusy THEN
		IF pFbGPInputRef^.bError THEN
			nStateA_InitTool := 99;
		ELSE
			nStateA_InitTool := 80;
		END_IF
		pFbGPInputRef^(bInit:= FALSE);
	END_IF
END_IF
END_ACTION

ACTION A_MeasurepH:
IF nStateA_MeasurepH = 0 THEN
	timer(IN:= TRUE,PT:= tTime);
	IF timer.Q THEN
		timer(IN:= FALSE);
		nStateA_MeasurepH := 80;
	END_IF
ELSIF nStateA_MeasurepH = 70 THEN
		timer(IN:= FALSE);
		nStateA_MeasurepH := 80;
END_IF
END_ACTION

ACTION A_Reset:
//Ist noch eine Aktion aktiv?
IF nStateA_ResetSpec = 0 THEN 
	(*IF bExpose THEN
		bExpose := FALSE;
		nStateA_Expose := 0;
	END_IF*)
	
	nStateA_ResetSpec := 80;
END_IF

SUPER^.A_Reset();
END_ACTION

ACTION A_Stop:
IF nStateA_Stop = 0 THEN

	IF bMeasurepH AND nStateA_MeasurepH < 70 THEN
		nStateA_MeasurepH := 70;
	END_IF
	
	nStateA_Stop := 1;
END_IF

SUPER^.A_Stop();
END_ACTION

METHOD FB_init : BOOL
VAR_INPUT
	bInitRetains : BOOL; // if TRUE, the retain variables are initialized (warm start / cold start)
	bInCopyCode : BOOL;  // if TRUE, the instance afterwards gets moved into the copy code (online change)
END_VAR
eObjectType := E_ObjectType.OBJECTTYPE_pHElectrode;
eObjectGroup := E_ObjectGroup.OBJECTGROUP_MzTool OR E_ObjectGroup.OBJECTGROUP_Device;
END_METHOD

METHOD M_AddChild : ERRORID
VAR_INPUT
	pObject : POINTER TO FB_Object;
	nSlotNr	: UINT;
	nIndex 	: INT;	
END_VAR
//Kann folgende Objekt-Typen aufnehmen
//pH-ElektrodeCAP
IF pObject > 0 THEN
	IF pObject^.P_eObjectType = E_ObjectType.OBJECTTYPE_pHElectrodeCap THEN
		M_AddChild := SUPER^.M_AddChild(pObject,nSlotNr,nIndex);
	ELSE
		M_AddChild := E_ErrorIdObjMgmt.ERRORID_InvalidParentObject;
	END_IF
ELSE
	M_AddChild := E_ErrorIdObjMgmt.ERRORID_InvalidParentObject;
END_IF
END_METHOD

METHOD M_AnswerSiblingForAction : ERRORID
VAR_INPUT
	eAction : E_Action;
END_VAR
IF eAction = E_Action.ACTION_MoveToTarget THEN
	IF pPiece > 0 THEN
		M_AnswerSiblingForAction := E_ErrorIdCmd.ERRORID_CapOnElectrode;
	END_IF
END_IF
END_METHOD

METHOD M_CancelAction
VAR_INPUT
	eAction : E_Action;
END_VAR
IF eAction = E_Action.ACTION_MeasurepH THEN
	IF bMeasurepH AND nStateA_MeasurepH < 70 THEN
		nStateA_MeasurepH := 70;
	END_IF
ELSE
	SUPER^.M_CancelAction(eAction);
END_IF
END_METHOD

METHOD M_CheckAction : ERRORID
VAR_INPUT
	refActionData 	: REFERENCE TO ST_ActionData;
	pCorrelObject	: POINTER TO FB_Object;
END_VAR

VAR
	pTarget 	: POINTER TO FB_TargetBase;
	pPieceEx	: POINTER TO FB_PieceBase;
END_VAR
CASE refActionData.eAction OF
	E_Action.ACTION_ExchangePiece:
		pTarget := fbObjectDirectory.M_GetObjPointer(refActionData.nTarget);
		IF pTarget^.P_eObjectType <> E_ObjectType.OBJECTTYPE_pHElectrodeCapRack THEN
			M_CheckAction := E_ErrorIdCmd.ERRORID_UnsuitableTarget;
		ELSE
			pPieceEx := pCorrelObject;
			IF pPieceEx^.P_eObjectType <> E_ObjectType.OBJECTTYPE_pHElectrodeCap THEN
				M_CheckAction := E_ErrorIdCmd.ERRORID_InvalidPieceType;
				RETURN;
			END_IF
			IF refActionData.aParams[2] = 0 THEN //Drop -> es muss ein Cap an pH-Elektrode sein
				IF pPiece = 0 THEN	 
					M_CheckAction := E_ErrorIdCmd.ERRORID_NoPieceOnTool;
					RETURN;	
				END_IF
			ELSIF refActionData.aParams[2] = 1 THEN //Take
				IF pPiece > 0 THEN	//Drop -> es darf kein Cap an pH-Elektrode sein
					M_CheckAction := E_ErrorIdCmd.ERRORID_PieceAlreadyOnTool;
					RETURN;
				END_IF
			ELSE
				M_CheckAction := E_ErrorIdCmd.ERRORID_InvalidCtrl;			
			END_IF
		END_IF
	E_Action.ACTION_MeasurepH:
		//1.Cap darf nicht am Tool sein
		IF pPiece > 0 THEN
			M_CheckAction := E_ErrorIdCmd.ERRORID_CapOnElectrode;
		END_IF	
ELSE
	M_CheckAction := SUPER^.M_CheckAction(refActionData, pCorrelObject);
END_CASE
END_METHOD

METHOD M_ExeAction : ERRORID
VAR_INPUT
	refActionData : REFERENCE TO ST_ActionData;	
END_VAR
IF NOT (eCurrentState = E_MachineState.MACHINESTATE_Idle OR
	eCurrentState = E_MachineState.MACHINESTATE_Active OR
	eCurrentState = E_MachineState.MACHINESTATE_Ready) THEN
	M_ExeAction := E_ErrorIdCmd.ERRORID_InvalidState;
	RETURN;
END_IF

CASE refActionData.eAction OF
	
	E_Action.ACTION_Init:
		IF NOT bInitAxis AND NOT bInitTool THEN
			bInitAxis := TRUE;
			bInitTool := TRUE;
			fbList.A_AddHeadValue( hList := hList, putValue := E_Action.ACTION_Init);	//InitAxis
			fbList.A_AddHeadValue( hList := hList, putValue := E_Action.ACTION_Init);	//InitTool
		ELSE
			RETURN;
		END_IF
		
	E_Action.ACTION_MeasurepH:
		IF NOT bMeasurepH THEN
			tTime := DINT_TO_TIME(refActionData.aParams[1]);
			fbList.A_AddHeadValue( hList := hList, putValue := E_Action.ACTION_MeasurepH);
			bMeasurepH := TRUE;
		ELSE
			M_ExeAction := E_ErrorIdCmd.ERRORID_BasicActionActive;
		END_IF
		
	ELSE
		M_ExeAction := SUPER^.M_ExeAction(refActionData);
		RETURN;
END_CASE
bBusy := TRUE;
eCurrentState := E_MachineState.MACHINESTATE_Active;
END_METHOD

METHOD M_GetAllProps : ERRORID
VAR_INPUT
	refCmdData : REFERENCE TO  ST_CmdData;
END_VAR
SUPER^.M_GetAllProps(refCmdData);
nCurrentPropIndex := nCurrentPropIndex + 1;
refCmdData.n32Data[nCurrentPropIndex] := nDigiOutChannelMz;
nCurrentPropIndex := nCurrentPropIndex + 1;
refCmdData.n32Data[nCurrentPropIndex] := nAnaInputChannelMz;
END_METHOD

METHOD M_SetAllProps : ERRORID
VAR_INPUT
	refCmdData : REFERENCE TO  ST_CmdData;
END_VAR
M_SetAllProps := SUPER^.M_SetAllProps(refCmdData);

IF M_SetAllProps > 0 THEN
	RETURN;
END_IF

//Digitaler Ausgang für Messverstärker
nCurrentPropIndex := nCurrentPropIndex + 1;
nSpecPropIndex := nCurrentPropIndex;
nDigiOutChannelMz := DINT_TO_USINT(refCmdData.n32Data[nCurrentPropIndex]);
IF NOT (nDigiOutChannelMz >= 1 AND nDigiOutChannelMz <= 7) THEN
	M_SetAllProps := E_ErrorIdObjMgmt.ERRORID_InvalidMzDOutChannel;
	RETURN;
END_IF

//Analoger Eingang für Messverstärker
nCurrentPropIndex := nCurrentPropIndex + 1;
nAnaInputChannelMz := DINT_TO_USINT(refCmdData.n32Data[nCurrentPropIndex]);
IF NOT (nAnaInputChannelMz >= 1 AND nAnaInputChannelMz <= 6) THEN
	M_SetAllProps := E_ErrorIdObjMgmt.ERRORID_InvalidAnaInputChannel;
	RETURN;
END_IF

pFbGPInputRef := ADR(pFbMultiZ^.aFbGPInputRef[nAnaInputChannelMz]);

nNoOfProps := nCurrentPropIndex + 1;
END_METHOD

METHOD M_SetSingleProp : ERRORID
VAR_INPUT
	refCmdData : REFERENCE TO  ST_CmdData;
END_VAR
IF nSpecPropIndex = refCmdData.aHeader[1] THEN
	IF NOT (refCmdData.n32Data[0] >= 1 AND refCmdData.n32Data[0] <= 7) THEN
		M_SetSingleProp := E_ErrorIdObjMgmt.ERRORID_InvalidMzDOutChannel;
		RETURN;
	END_IF
	nDigiOutChannelMz := DINT_TO_USINT(refCmdData.n32Data[0]);
ELSIF (nSpecPropIndex + 1) = refCmdData.aHeader[1] THEN
	IF NOT (refCmdData.n32Data[0] >= 1 AND refCmdData.n32Data[0] <= 6) THEN
		M_SetSingleProp := E_ErrorIdObjMgmt.ERRORID_InvalidAnaInputChannel;
		RETURN;
	END_IF	
	nAnaInputChannelMz := DINT_TO_USINT(refCmdData.n32Data[0]);
	pFbGPInputRef := ADR(pFbMultiZ^.aFbGPInputRef[nAnaInputChannelMz]);
ELSE
	M_SetSingleProp := SUPER^.M_SetSingleProp(refCmdData);
END_IF
END_METHOD

PROPERTY P_nCurrentpHValue : DINT
GET
P_nCurrentpHValue := REAL_TO_DINT(rCurrentpHValue * 1000.0);
END_GET
END_PROPERTY

PROPERTY P_rToolRadius : REAL
GET
VAR
	stDim : ST_3DDimension;
END_VAR
P_rToolRadius := 3000.0;
END_GET
END_PROPERTY

END_FUNCTION_BLOCK

// ---- Hardware/XYDrive/CoupleYY.TcPOU
PROGRAM CoupleYY
VAR_INPUT
	bCouple : BOOL;
	bExecute : BOOL;
END_VAR
VAR_OUTPUT
	bBusy : BOOL;
	bError : BOOL;
	nErrorID : ERRORID;
END_VAR
VAR
	nState : USINT;
	fbMcGearIn	: Tc2_MC2.MC_GearIn;
	fbMcGearOut	: Tc2_MC2.MC_GearOut;
END_VAR

//AxisRefY1 ist bei Plattform D immer unten
//AxisRefY2 ist bei Plattform D immer oben
//Grundsätzlich muss hier nicht überprüft werden, ob es Plattform C oder D ist, denn es würde ohnehin zu einem Fehler kommen
IF bExecute THEN
	IF nState = 0 THEN
		//Status überprüfen
		//1. Beide Achsen müssen initialisiert sein
		//2. Beide Achsen dürfen nicht Busy oder im Error sein
		IF AxisRefY1.Status.Error OR AxisRefY2.Status.Error OR AxisRefY1.Status.Moving OR AxisRefY2.Status.Moving THEN
			bError := TRUE;
			nErrorID := E_ErrorIdCmd.ERRORID_AxisStillBusy;
			RETURN;
		END_IF
		IF NOT(AxisRefY1.Status.Homed AND AxisRefY2.Status.Homed) THEN
			bError := TRUE;
			nErrorID := E_ErrorIdCmd.ERRORID_DeviceNotInitialized;
			RETURN;
		END_IF
		IF bCouple THEN	//Ankoppeln - Achse darf noch nicht gekoppelt sein
			IF AxisRefY1.Status.Coupled THEN
				bError := TRUE;
				{warning 'Implement right ErrorID}
				nErrorID := E_ErrorIdCmd.ERRORID_X2AxisNotCoupled;
				RETURN;
			END_IF
			nState := 1;
		ELSE //Auskopplen - Achse muss eingekoppelt sein
			IF NOT AxisRefY1.Status.Coupled THEN
				bError := TRUE;
				{warning 'Implement right ErrorID}
				nErrorID := E_ErrorIdCmd.ERRORID_X2AxisNotCoupled;
				RETURN;
			END_IF
			nState := 2;
		END_IF
		bBusy := TRUE;
	END_IF
	
	IF nState = 1 THEN	//Ankoppeln
		fbMcGearIn(Master:= AxisRefY2, Slave:= AxisRefY1, Execute:= TRUE, RatioNumerator:= 1.0,	RatioDenominator:= 1);
		IF NOT fbMcGearIn.Busy THEN
			IF fbMcGearIn.Error THEN
				bError := TRUE;
				nErrorID := UDINT_TO_UINT(fbMcGearIn.ErrorID);
				nState := 99;
			END_IF
			bBusy := FALSE;
			fbMcGearIn(Master:= AxisRefY2, Slave:= AxisRefY1, Execute:= FALSE);
		END_IF
	ELSIF nState = 2 THEN //Abkoppeln
		fbMcGearOut(Slave:= AxisRefY1, Execute:= TRUE);
		IF NOT fbMcGearOut.Busy THEN
			IF fbMcGearOut.Error THEN
				bError := TRUE;
				nErrorID := UDINT_TO_UINT(fbMcGearOut.ErrorID);
				nState := 99;				
			END_IF
			bBusy := FALSE;
			fbMcGearOut(Slave:= AxisRefY1, Execute:= FALSE);
		END_IF
	END_IF

ELSE
	nState := 0;
	bBusy := FALSE;
	bError := FALSE;
	nErrorID	:= 0;
END_IF

END_PROGRAM

// ---- Sequence/F_SetFollowerStep.TcPOU
FUNCTION F_SetFollowerStep : ERRORID
VAR_INPUT
	pStep			: POINTER TO ST_Step;
	nFollowerStepNr : UINT;
END_VAR
VAR
	i : USINT;
	nMaxFollowers : USINT;
END_VAR

IF pStep > 0 THEN
	IF nFollowerStepNr > 0 THEN
		nMaxFollowers := UINT_TO_USINT(SIZEOF (pStep^.aFollower) / 2);
		FOR i:= 0 TO (nMaxFollowers - 1) BY 1 DO
			IF pStep^.aFollower[i] = 0 THEN
				pStep^.aFollower[i] := nFollowerStepNr;
				RETURN;
			END_IF
		END_FOR
		F_SetFollowerStep := E_ErrorIdCmd.ERRORID_NoOfFollowerStepsExeeded;		
	ELSE
		F_SetFollowerStep := E_ErrorIdCmd.ERRORID_InvalidStepNr;
	END_IF
END_IF

END_FUNCTION

// ---- Sequence/FB_CondiStepReady.TcPOU
{attribute 'enable_dynamic_creation'}
FUNCTION_BLOCK FB_CondiStepReady EXTENDS FB_CondiBase
VAR_INPUT
END_VAR
VAR_OUTPUT
END_VAR
VAR
	pStep : POINTER TO ST_Step;
END_VAR

METHOD M_Check : BYTE
VAR_INPUT
	nPreResult : BYTE;
END_VAR

VAR
	bResult : BOOL;
END_VAR
//es wird nur Bit0 entsprechend verknüpft
//Bit1 steht für "Cancel" und wird derzeit nur FB_CondiStepResult verküpft

IF eCondiOperator = E_LogicOperator.LOGIC_OP_AND THEN
	nPreResult.0 := nPreResult.0 AND (pStep^.eState = E_StepState.STEPSTATUS_Ready);
ELSIF eCondiOperator = E_LogicOperator.LOGIC_OP_OR THEN
	nPreResult.0 := nPreResult.0 OR (pStep^.eState = E_StepState.STEPSTATUS_Ready);
END_IF

IF pNextCondi > 0 THEN
	M_Check := pNextCondi^.M_Check(nPreResult);
ELSE
	M_Check  := nPreResult;
END_IF
END_METHOD

PROPERTY P_pStep : POINTER TO ST_Step
SET
pStep := P_pStep;
END_SET
END_PROPERTY

END_FUNCTION_BLOCK

// ---- Sequence/FB_CondiProcessData.TcPOU
{attribute 'enable_dynamic_creation'}
FUNCTION_BLOCK FB_CondiProcessData EXTENDS FB_CondiBase
VAR_INPUT
END_VAR
VAR_OUTPUT
END_VAR
VAR
	eProcDataType : E_ProcDataType;
	iDevice		  : I_Device;
	nCompareValue : DINT;
END_VAR

PROPERTY P_iDevice : I_Device
SET
iDevice := P_iDevice;
END_SET
END_PROPERTY

PROPERTY P_nValue : DINT
SET
nCompareValue := P_nValue;
END_SET
END_PROPERTY

METHOD M_Check : BYTE
VAR_INPUT
	nPreResult : BYTE;
END_VAR

VAR
	bResult			: BOOL;
	nCurrentValue	: DINT;
END_VAR
nCurrentValue := iDevice.M_GetProcData(eProcDataType);

IF eCondition = E_Condition.CONDITION_ProcessVarLEQ THEN
	IF nCurrentValue <= nCompareValue THEN
		bResult := TRUE;
	END_IF
ELSIF eCondition = E_Condition.CONDITION_ProcessVarGEQ THEN
	IF nCurrentValue >= nCompareValue THEN
		bResult := TRUE;
	END_IF	
END_IF

//es wird nur Bit0 entsprechend verknüpft
//Bit1 steht für "Cancel" und wird derzeit nur FB_CondiStepResult verküpft
IF eCondiOperator = E_LogicOperator.LOGIC_OP_AND THEN
	nPreResult.0 := nPreResult.0 AND bResult;
ELSIF eCondiOperator = E_LogicOperator.LOGIC_OP_OR THEN
	nPreResult.0 := nPreResult.0 OR bResult;
END_IF

IF pNextCondi > 0 THEN
	M_Check := pNextCondi^.M_Check(nPreResult);
ELSE
	M_Check  := nPreResult;
END_IF
END_METHOD

PROPERTY P_eProcDataType : E_ProcDataType
SET
eProcDataType := P_eProcDataType;
END_SET
END_PROPERTY

END_FUNCTION_BLOCK

// ---- Sequence/FB_CondiStepResult.TcPOU
{attribute 'enable_dynamic_creation'}
FUNCTION_BLOCK FB_CondiStepResult EXTENDS FB_CondiBase
VAR_INPUT
END_VAR
VAR_OUTPUT
END_VAR
VAR
	pStep 			: POINTER TO ST_Step;
	eCompareOperator: E_CompOperator;
	nCompareValue 	: DINT;
END_VAR

PROPERTY P_eCompareOperator : E_CompOperator
GET
P_eCompareOperator := eCompareOperator;
END_GET
SET
eCompareOperator := P_eCompareOperator;
END_SET
END_PROPERTY

PROPERTY P_nCompareValue : DINT
SET
nCompareValue := P_nCompareValue;
END_SET
END_PROPERTY

PROPERTY P_pStep : POINTER TO ST_Step
SET
pStep := P_pStep;
END_SET
END_PROPERTY

METHOD M_Check : BYTE
VAR_INPUT
	nPreResult : BYTE;
END_VAR

VAR
	bCancel : BOOL := TRUE;
END_VAR
IF pStep^.bActionResultIsValid  AND (pStep^.eState = E_StepState.STEPSTATUS_Ready) THEN
	IF eCondiOperator = E_LogicOperator.LOGIC_OP_AND THEN
		//nPreResult.0 := nPreResult.0 AND TRUE;
	ELSIF eCondiOperator = E_LogicOperator.LOGIC_OP_OR THEN
		nPreResult.0 := TRUE;
	END_IF
	
	IF nPreResult.0 THEN
		CASE eCompareOperator OF
			E_CompOperator.COMP_OP_GT:	//>
				IF pStep^.nActionResult > nCompareValue THEN
					bCancel := FALSE;
				END_IF
			E_CompOperator.COMP_OP_LT:	//<
				IF pStep^.nActionResult < nCompareValue THEN
					bCancel := FALSE;
				END_IF
			E_CompOperator.COMP_OP_GE:	//>=
				IF pStep^.nActionResult >= nCompareValue THEN
					bCancel := FALSE;
				END_IF
			E_CompOperator.COMP_OP_LE:	//<=
				IF pStep^.nActionResult <= nCompareValue THEN
					bCancel := FALSE;
				END_IF
			E_CompOperator.COMP_OP_EQ:	//=
				IF pStep^.nActionResult = nCompareValue THEN
					bCancel := FALSE;
				END_IF
		END_CASE
		
		IF eCondiOperator = E_LogicOperator.LOGIC_OP_AND THEN
			nPreResult.1 := nPreResult.1 OR bCancel;
		ELSIF eCondiOperator = E_LogicOperator.LOGIC_OP_OR THEN
			IF NOT bCancel THEN
				nPreResult.1 := FALSE;
			END_IF
		END_IF
		
		IF pNextCondi > 0 THEN
			M_Check := pNextCondi^.M_Check(nPreResult);
		ELSE
			M_Check  := nPreResult;
		END_IF		
	END_IF
END_IF
END_METHOD

END_FUNCTION_BLOCK

// ---- GCode/FB_FastMFunc.TcPOU
FUNCTION_BLOCK FB_FastMFunc
VAR_INPUT
	bStop : BOOL;
END_VAR
VAR_OUTPUT
	bBusy				: BOOL;
	bError				: BOOL;
	nErrorId			: ERRORID;	
END_VAR
VAR_IN_OUT
	stGCodeRef			: ST_GCodeRef;
END_VAR
VAR
	fbItpResetFastMFuncEx100	: Tc2_NCI.ItpResetFastMFuncEx;
	fbItpResetFastMFuncEx104	: Tc2_NCI.ItpResetFastMFuncEx;
	fbItpResetFastMFuncEx105	: Tc2_NCI.ItpResetFastMFuncEx;
	fbItpGoAhead				: Tc2_NCI.ItpGoAhead;
	
	fbAdsRead1					: ADSREAD;
	fbAdsRead2					: ADSREAD;
	
	stCurrentPos				: ST_3DPoint;
	
	nStateA_FastMFunk100: USINT;
	
	rTrigM104			: R_TRIG;
	rTrigM105			: R_TRIG;
	
	eCurModalGeoType	: E_ModalGeoTypes;
	aTechnoData			: ARRAY[0..1] OF UDINT;
	alXYTargetPos		: ARRAY[0..2] OF LREAL;
	alQ1TargetPos		: ARRAY[0..4] OF LREAL;
	
	nCyclCounter		: USINT;
	nCyclThreshold		: USINT := 20;
	
	stActionDataMoveZ	: ST_ActionData;
	nStateA_MoveZ		: USINT;
	
	stError 			: ST_Error := (POU := E_POU.POU_GCode);
END_VAR

fbItpResetFastMFuncEx100(sNciToPlc:= stGCodeRef.sNciToPlc);
IF fbItpResetFastMFuncEx100.bExecute AND NOT fbItpResetFastMFuncEx100.bBusy THEN
	fbItpResetFastMFuncEx100(bExecute:= FALSE, nMFuncNo:= 100 , sNciToPlc:= stGCodeRef.sNciToPlc);
END_IF

fbItpResetFastMFuncEx104(sNciToPlc:= stGCodeRef.sNciToPlc);
IF fbItpResetFastMFuncEx104.bExecute AND NOT fbItpResetFastMFuncEx104.bBusy THEN
	fbItpResetFastMFuncEx104(bExecute:= FALSE, nMFuncNo:= 104 , sNciToPlc:= stGCodeRef.sNciToPlc);
END_IF

fbItpResetFastMFuncEx105(sNciToPlc:= stGCodeRef.sNciToPlc);
IF fbItpResetFastMFuncEx105.bExecute AND NOT fbItpResetFastMFuncEx104.bBusy THEN
	fbItpResetFastMFuncEx105(bExecute:= FALSE, nMFuncNo:= 105 , sNciToPlc:= stGCodeRef.sNciToPlc);
END_IF

fbItpGoAhead();
IF fbItpGoAhead.bExecute AND NOT fbItpGoAhead.bBusy THEN
	fbItpGoAhead(bExecute:= FALSE);
END_IF

//***************************M100 MoveZ*************************************
IF ItpIsFastMFunc(100,stGCodeRef.sNciToPlc) THEN	//G00,G01 Q1=x M100 @717
	CASE nStateA_FastMFunk100 OF	//20Zyklen warten, damit Technologiedaten aktuell
		0:	nCyclCounter := nCyclCounter + 1;
			IF nCyclCounter = nCyclThreshold THEN
				nCyclCounter := 0;
				nStateA_FastMFunk100 := 10;
			END_IF
		
		10:	//Technologiedaten lesen (muss unbegingt vor dem Auslesen der Z-Position erfolgen)
			//zumindest sollte vor dem Auslesen der Z-Position noch ein Zyklus stattfinden
			//NC-Override auf "0" setzen damit XY noch nicht losfahren, bis ZMove beginnt
			stGCodeRef.lrNcOverride := 0.0;
			ItpSetOverridePercent(stGCodeRef.lrNcOverride,stGCodeRef.sPlcToNci);
			
			fbAdsRead1(PORT:= 501, IDXGRP:= 16#2100 + ItpGetChannelId(stGCodeRef.sNciToPlc), IDXOFFS:= 16#13 ,
						LEN:= SIZEOF(aTechnoData), DESTADDR:= ADR(aTechnoData), READ:= TRUE);
			IF NOT fbAdsRead1.BUSY THEN
				IF fbAdsRead1.ERR THEN
					bError := TRUE;
					nErrorId := UDINT_TO_UINT(fbAdsRead1.ERRID);
				ELSE
					IF bStop THEN
						nStateA_FastMFunk100 := 0;
						bBusy := FALSE;
					ELSE
						nStateA_FastMFunk100 := 20;	
					END_IF
				END_IF
				fbAdsRead1(READ:=FALSE);
			END_IF
			
		20:	//Positionen aus NCI lesen
			//TargetPos XY
			nStateA_FastMFunk100 := 30;
			fbAdsRead1(PORT:= 501, IDXGRP:= 16#3100 + ItpGetGroupId(stGCodeRef.sNciToPlc), IDXOFFS:= 16#530 ,	
					LEN:= SIZEOF(alXYTargetPos), DESTADDR:= ADR(alXYTargetPos), READ:= TRUE);

			//TargetPos Q1
			fbAdsRead2(PORT:= 501, IDXGRP:= 16#3100 + ItpGetGroupId(stGCodeRef.sNciToPlc), IDXOFFS:= 16#531 ,	
					LEN:= SIZEOF(alQ1TargetPos), DESTADDR:= ADR(alQ1TargetPos), READ:= TRUE);

			IF fbAdsRead1.ERR THEN
				bError := TRUE;
				nErrorId := UDINT_TO_UINT(fbAdsRead1.ERRID);
				fbAdsRead1(READ:=FALSE);
			END_IF
			

			IF fbAdsRead2.ERR THEN
				bError := TRUE;
				nErrorId := UDINT_TO_UINT(fbAdsRead1.ERRID);
				fbAdsRead2(READ:=FALSE);
			END_IF
			
			IF NOT (fbAdsRead1.BUSY OR fbAdsRead2.BUSY) THEN
				IF bStop THEN
					nStateA_FastMFunk100 := 0;
					bBusy := FALSE;
				END_IF
				fbAdsRead1(READ:=FALSE);
				fbAdsRead2(READ:=FALSE);
			ELSE
				nStateA_FastMFunk100 := 20;
			END_IF
			
		30:	
			eCurModalGeoType := aTechnoData[1];
			stActionDataMoveZ.aParams[1] := E_MoveMode.MODE_AbsWithOffset;
			stCurrentPos := stGCodeRef.pCurrentTool^.P_stCurrentPosTotal;
			//befindet sich aktuelle XY-Position außerhalb des GCode-Druckbereichs, dann Fehler werfen
			IF NOT stGCodeRef.fbLimitCuboid.M_IsPointInnerXY(stCurrentPos) THEN
				nStateA_FastMFunk100 := 0;
				stGCodeRef.lrNcOverride := 100.0;
				bBusy := FALSE;
				bError := TRUE;
				nErrorId := E_ErrorIdGCode.ERRORID_ZMoveOutsidePrintArea;
				RETURN;
			END_IF
			
			CASE eCurModalGeoType OF
				E_ModalGeoTypes.MODALGEOTYPE_G0:	//Eilgang
					stActionDataMoveZ.aParams[3] := -1;	//max Speed
					A_MoveZ();
					nStateA_FastMFunk100 := 40;
				E_ModalGeoTypes.MODALGEOTYPE_G01,E_ModalGeoTypes.MODALGEOTYPE_G02,E_ModalGeoTypes.MODALGEOTYPE_G03:
					stActionDataMoveZ.aParams[3] := LREAL_TO_DINT(stGCodeRef.sNciToPlc.DoubleParams[0] * 1000); (*programmierte Geschwindigkeit des aktuellen Segments*)
					IF stActionDataMoveZ.aParams[3] = 0 THEN
						stGCodeRef.lrNcOverride := 100.0;
						ItpSetOverridePercent(stGCodeRef.lrNcOverride,stGCodeRef.sPlcToNci);
						fbItpGoAhead(bExecute:= TRUE, nChnId:= ItpGetChannelId(stGCodeRef.sNciToPlc));
						nStateA_MoveZ := 0;
						nStateA_FastMFunk100 := 0;
						fbItpResetFastMFuncEx100(bExecute:= TRUE, nMFuncNo:= 100 , sNciToPlc:= stGCodeRef.sNciToPlc);
					ELSE
						A_MoveZ();
						nStateA_FastMFunk100 := 40;
					END_IF
			ELSE
				nStateA_FastMFunk100 := 0;
				fbItpResetFastMFuncEx100(bExecute:= TRUE, nMFuncNo:= 100 , sNciToPlc:= stGCodeRef.sNciToPlc);
				fbItpGoAhead(bExecute:= TRUE, nChnId:= ItpGetChannelId(stGCodeRef.sNciToPlc));
			END_CASE
					
		40:	//MoveZ ready?
			A_MoveZ();
			stGCodeRef.lrNcOverride := 100.0;
			ItpSetOverridePercent(stGCodeRef.lrNcOverride,stGCodeRef.sPlcToNci);
			IF nStateA_MoveZ >= 80 THEN
				IF nStateA_MoveZ >= 99 THEN
					bError := TRUE;
				ELSE
					IF bStop THEN
						bBusy := FALSE;
					ELSE
						fbItpGoAhead(bExecute:= TRUE, nChnId:= ItpGetChannelId(stGCodeRef.sNciToPlc));
					END_IF
				END_IF
				nStateA_MoveZ := 0;
				nStateA_FastMFunk100 := 0;
				fbItpResetFastMFuncEx100(bExecute:= TRUE, nMFuncNo:= 100 , sNciToPlc:= stGCodeRef.sNciToPlc);
			END_IF
	END_CASE
END_IF

IF ItpIsFastMFunc(150,stGCodeRef.sNciToPlc) THEN	//M150 DigiOut On
	bTrigger2 := TRUE;
END_IF

IF ItpIsFastMFunc(151,stGCodeRef.sNciToPlc) THEN	//M151 DigiOut Off
	bTrigger2 := FALSE;
END_IF

//***************************M104 PrintActorOff* Channel1****************************************
rTrigM104(CLK:= ItpIsFastMFunc(104,stGCodeRef.sNciToPlc));
IF rTrigM104.Q THEN
	//Abhängig vom Tool den entsprechenden PrintActor ausschalten
	M_StopPrintAction(stGCodeRef.pCurrentTool,1);
	stGCodeRef.aToolTable[stGCodeRef.sNciToPlc.Tool].bIsInAction1 := FALSE;
	fbItpResetFastMFuncEx104(bExecute:= TRUE, nMFuncNo:= 104 , sNciToPlc:= stGCodeRef.sNciToPlc);
END_IF

//***************************M105 PrintActorOff* Channel2****************************************
rTrigM105(CLK:= ItpIsFastMFunc(105,stGCodeRef.sNciToPlc));
IF rTrigM105.Q THEN
	M_StopPrintAction(stGCodeRef.pCurrentTool,2);
	stGCodeRef.aToolTable[stGCodeRef.sNciToPlc.Tool].bIsInAction2 := FALSE;
	fbItpResetFastMFuncEx105(bExecute:= TRUE, nMFuncNo:= 105 , sNciToPlc:= stGCodeRef.sNciToPlc);
END_IF

IF NOT bStop THEN
	IF ItpIsFastMFunc(100,stGCodeRef.sNciToPlc) OR ItpIsFastMFunc(104,stGCodeRef.sNciToPlc) OR
		ItpIsFastMFunc(105,stGCodeRef.sNciToPlc) OR fbItpGoAhead.bExecute THEN
		bBusy := TRUE;
	ELSE
		bBusy := FALSE;
	END_IF	
END_IF

ACTION A_MoveZ:
stError.POUState := nStateA_MoveZ;

CASE nStateA_MoveZ OF
	0:
		IF stGCodeRef.pCurrentTool = 0 THEN
			stError.Cmd := E_Action.ACTION_MoveZ;
			stError.ErrorId := E_ErrorIdGCode.ERRORID_NoSelectedTool;
			nStateA_MoveZ := 99;
		ELSE
			stActionDataMoveZ.eAction := E_Action.ACTION_MoveZ;
			
			IF stActionDataMoveZ.aParams[3] > REAL_TO_DINT(stGCodeRef.pCurrentTool^.M_GetMaxSpeed(E_MoveDirection.DIRECTION_ZPLUS)) THEN
				stActionDataMoveZ.aParams[3]:= -1; //MaxSpeed Z
			END_IF
			
			//MoveMode = absolut ? -> Nullpunktverschiebung verrechnen
			IF stActionDataMoveZ.aParams[1] = E_MoveMode.MODE_AbsWithOffset THEN
				stActionDataMoveZ.aParams[2] := LREAL_TO_DINT((stGCodeRef.sZeroShiftDesc.fShiftZ + alQ1TargetPos[0]) * 1000.0);
			ELSE
				stActionDataMoveZ.aParams[2] := LREAL_TO_DINT(alQ1TargetPos[0]);
			END_IF
			
			stError.ErrorId := stGCodeRef.pCurrentTool^.M_ExeAction(stActionDataMoveZ);
			
			IF stError.ErrorId > 0 THEN
				nStateA_MoveZ := 99;
			ELSE
				nStateA_MoveZ := 1;
			END_IF			
		END_IF
	

	1:	//Move ready?
		IF NOT stGCodeRef.pCurrentTool^.M_GetActionBusy(E_Action.ACTION_MoveZ) THEN
			IF stGCodeRef.pCurrentTool^.P_bError THEN
				stError.ErrorId := stGCodeRef.pCurrentTool^.P_nErrorId;
				nStateA_MoveZ := 99;
			ELSE
				nStateA_MoveZ := 80;
			END_IF
		END_IF
END_CASE

IF nStateA_MoveZ = 99 THEN
	stError.POUAction := E_POUACT.POUACT_A_MoveZ;
	fbErrorList.M_Add(stError);	
END_IF
END_ACTION

METHOD M_Reset
VAR_INPUT
END_VAR
fbItpResetFastMFuncEx100(bExecute:= FALSE, sNciToPlc:= stGCodeRef.sNciToPlc);
fbItpResetFastMFuncEx104(bExecute:= FALSE, sNciToPlc:= stGCodeRef.sNciToPlc);
fbItpResetFastMFuncEx105(bExecute:= FALSE, sNciToPlc:= stGCodeRef.sNciToPlc);
fbItpGoAhead(bExecute:= FALSE);
nStateA_FastMFunk100 := 0;
nStateA_MoveZ := 0;
nCyclCounter := 0;
bBusy := FALSE;
bError := FALSE;
nErrorId := 0;
END_METHOD

METHOD M_StopPrintAction : ERRORID
VAR_INPUT
	pTool	: POINTER TO FB_MzTool;
	nChannel : DINT;
END_VAR

VAR
	stAction : ST_ActionData;
	pMultiCartHolder : POINTER TO FB_MultiCartHolder;
END_VAR
IF pTool > 0 THEN
	CASE pTool^.P_eObjectType OF
		E_ObjectType.OBJECTTYPE_CartDispenser,
		E_ObjectType.OBJECTTYPE_CartDispStirrer:
			stAction.eAction := E_Action.ACTION_SwitchPressure;
			pTool^.M_ExeAction(stAction);
			stAction.eAction := E_Action.ACTION_Expose;
			pTool^.M_ExeAction(stAction);
		E_ObjectType.OBJECTTYPE_MultiCartHolder:
			pMultiCartHolder := pTool;
			//In Abhängigkeit vom Channel auf die einzelnen Dispenser anwenden
			stAction.eAction := E_Action.ACTION_SwitchPressure;
			CASE nChannel OF
				0:	pMultiCartHolder^.M_ExeAction(stAction);
				
				1:	IF pMultiCartHolder^.P_pCartDispenser1 > 0 THEN
						pMultiCartHolder^.P_pCartDispenser1^.M_ExeAction(stAction);
					END_IF
					
				2:	IF pMultiCartHolder^.P_pCartDispenser2 > 0 THEN
						pMultiCartHolder^.P_pCartDispenser2^.M_ExeAction(stAction);
					END_IF
					
				3:	IF pMultiCartHolder^.P_pCartDispenser3 > 0 THEN
						pMultiCartHolder^.P_pCartDispenser3^.M_ExeAction(stAction);
					END_IF
			END_CASE
		E_ObjectType.OBJECTTYPE_HybridDispenser:
			stAction.eAction := E_Action.ACTION_BasicDispense;	
			pTool^.M_ExeAction(stAction);
		E_ObjectType.OBJECTTYPE_DeloDot, E_ObjectType.OBJECTTYPE_PiezoPip, E_ObjectType.OBJECTTYPE_TwinPiezoHolder, E_ObjectType.OBJECTTYPE_SolenoidPip,
			E_ObjectType.OBJECTTYPE_VermesDisp:
			stAction.eAction := E_Action.ACTION_DispenseDrops;
			//restliche Paremeter sind sowieso "0"
			pTool^.M_ExeAction(stAction);
		E_ObjectType.OBJECTTYPE_Exposure:
			stAction.eAction := E_Action.ACTION_Expose;
			pTool^.M_ExeAction(stAction);
		E_ObjectType.OBJECTTYPE_PassivPip:
			pTool^.M_CancelAction(E_Action.ACTION_Dispense);
		E_ObjectType.OBJECTTYPE_Extruder:
			stAction.eAction := E_Action.ACTION_Extrude;
			pTool^.M_ExeAction(stAction);
		E_ObjectType.OBJECTTYPE_TwinExtruder:
			stAction.eAction := E_Action.ACTION_Extrude;
			pTool^.M_ExeAction(stAction);
	ELSE
		RETURN;
	END_CASE
END_IF
END_METHOD

END_FUNCTION_BLOCK

